	bStn3MegasonicOnOffLevel[1]:=FALSE;
	bStn3MegasonicOnOffLevel[2]:=FALSE;
	bStn3MegasonicOnOffLevel[4]:=FALSE;
	bStn3MegasonicOnOffLevel[5]:=FALSE;
END_IF

bResetMegasonicPower_RE[4](CLK:=bStn3MegasonicOnOffLevel[4]  , Q=> );	
IF bResetMegasonicPower_RE[4].Q THEN
	ARwDO[eY11104_Stn03MegasonicGenerator01Power01].15 :=FALSE;
	ARwDO[eY11105_Stn03MegasonicGenerator01Power02].15 :=FALSE;
	ARwDO[eY11106_Stn03MegasonicGenerator01Power03].15 :=FALSE;
	ARwDO[eY11108_Stn03MegasonicGenerator01Power05].15 :=FALSE;
	
	ARwDO[eY11110_Stn03MegasonicGenerator02Power01].15 :=FALSE;
	ARwDO[eY11111_Stn03MegasonicGenerator02Power02].15 :=FALSE;
	ARwDO[eY11112_Stn03MegasonicGenerator02Power03].15 :=FALSE;
	ARwDO[eY11114_Stn03MegasonicGenerator02Power05].15 :=FALSE;
	
	bStn3MegasonicOnOffLevel[1]:=FALSE;
	bStn3MegasonicOnOffLevel[2]:=FALSE;
	bStn3MegasonicOnOffLevel[3]:=FALSE;
	bStn3MegasonicOnOffLevel[5]:=FALSE;
END_IF

bResetMegasonicPower_RE[5](CLK:=bStn3MegasonicOnOffLevel[5]  , Q=> );	
IF bResetMegasonicPower_RE[5].Q THEN
	ARwDO[eY11104_Stn03MegasonicGenerator01Power01].15 :=FALSE;
	ARwDO[eY11105_Stn03MegasonicGenerator01Power02].15 :=FALSE;
	ARwDO[eY11106_Stn03MegasonicGenerator01Power03].15 :=FALSE;
	ARwDO[eY11107_Stn03MegasonicGenerator01Power04].15 :=FALSE;
	
	ARwDO[eY11110_Stn03MegasonicGenerator02Power01].15 :=FALSE;
	ARwDO[eY11111_Stn03MegasonicGenerator02Power02].15 :=FALSE;
	ARwDO[eY11112_Stn03MegasonicGenerator02Power03].15 :=FALSE;
	ARwDO[eY11107_Stn03MegasonicGenerator01Power04].15 :=FALSE;
	
	bStn3MegasonicOnOffLevel[1]:=FALSE;
	bStn3MegasonicOnOffLevel[2]:=FALSE;
	bStn3MegasonicOnOffLevel[3]:=FALSE;
	bStn3MegasonicOnOffLevel[4]:=FALSE;
END_IF	


//////// Station 6 Megasonic 
bResetMegasonicPower_RE[6](CLK:=bStn6MegasonicOnOffLevel[1]  , Q=> );	
IF bResetMegasonicPower_RE[6].Q THEN
	ARwDO[eY12004_Stn06MegasonicGenerator01Power02].15 :=FALSE;
	ARwDO[eY12005_Stn06MegasonicGenerator01Power03].15 :=FALSE;
	ARwDO[eY12006_Stn06MegasonicGenerator01Power04].15 :=FALSE;
	ARwDO[eY12007_Stn06MegasonicGenerator01Power05].15 :=FALSE;
	
	ARwDO[eY12010_Stn06MegasonicGenerator02Power02].15 :=FALSE;
	ARwDO[eY12011_Stn06MegasonicGenerator02Power03].15 :=FALSE;
	ARwDO[eY12012_Stn06MegasonicGenerator02Power04].15 :=FALSE;
	ARwDO[eY12013_Stn06MegasonicGenerator02Power05].15 :=FALSE;
	
	bStn6MegasonicOnOffLevel[2] := FALSE;
	bStn6MegasonicOnOffLevel[3] := FALSE;
	bStn6MegasonicOnOffLevel[4] := FALSE;
	bStn6MegasonicOnOffLevel[5] := FALSE;
	
END_IF

bResetMegasonicPower_RE[7](CLK:=bStn6MegasonicOnOffLevel[2]  , Q=> );	
IF bResetMegasonicPower_RE[7].Q THEN
	ARwDO[eY12003_Stn06MegasonicGenerator01Power01].15 :=FALSE;
	ARwDO[eY12005_Stn06MegasonicGenerator01Power03].15 :=FALSE;
	ARwDO[eY12006_Stn06MegasonicGenerator01Power04].15 :=FALSE;
	ARwDO[eY12007_Stn06MegasonicGenerator01Power05].15 :=FALSE;
	
	ARwDO[eY12009_Stn06MegasonicGenerator02Power01].15 :=FALSE;
	ARwDO[eY12011_Stn06MegasonicGenerator02Power03].15 :=FALSE;
	ARwDO[eY12012_Stn06MegasonicGenerator02Power04].15 :=FALSE;
	ARwDO[eY12013_Stn06MegasonicGenerator02Power05].15 :=FALSE;
	
	bStn6MegasonicOnOffLevel[1] := FALSE;
	bStn6MegasonicOnOffLevel[3] := FALSE;
	bStn6MegasonicOnOffLevel[4] := FALSE;
	bStn6MegasonicOnOffLevel[5] := FALSE;
END_IF
	
	


bResetMegasonicPower_RE[8](CLK:=bStn6MegasonicOnOffLevel[3]  , Q=> );	
IF bResetMegasonicPower_RE[8].Q THEN
	ARwDO[eY12003_Stn06MegasonicGenerator01Power01].15 :=FALSE;
	ARwDO[eY12004_Stn06MegasonicGenerator01Power02].15 :=FALSE;
	ARwDO[eY12006_Stn06MegasonicGenerator01Power04].15 :=FALSE;
	ARwDO[eY12007_Stn06MegasonicGenerator01Power05].15 :=FALSE;
	
	ARwDO[eY12009_Stn06MegasonicGenerator02Power01].15 :=FALSE;
	ARwDO[eY12010_Stn06MegasonicGenerator02Power02].15 :=FALSE;
	ARwDO[eY12012_Stn06MegasonicGenerator02Power04].15 :=FALSE;
	ARwDO[eY12013_Stn06MegasonicGenerator02Power05].15 :=FALSE;
	
	bStn6MegasonicOnOffLevel[1] := FALSE;
	bStn6MegasonicOnOffLevel[2] := FALSE;
	bStn6MegasonicOnOffLevel[4] := FALSE;
	bStn6MegasonicOnOffLevel[5] := FALSE;
END_IF

	

bResetMegasonicPower_RE[9](CLK:=bStn6MegasonicOnOffLevel[4]  , Q=> );	
IF bResetMegasonicPower_RE[9].Q THEN
	ARwDO[eY12003_Stn06MegasonicGenerator01Power01].15 :=FALSE;
	ARwDO[eY12004_Stn06MegasonicGenerator01Power02].15 :=FALSE;
	ARwDO[eY12005_Stn06MegasonicGenerator01Power03].15 :=FALSE;
	ARwDO[eY12007_Stn06MegasonicGenerator01Power05].15 :=FALSE;
	
	ARwDO[eY12009_Stn06MegasonicGenerator02Power01].15 :=FALSE;
	ARwDO[eY12010_Stn06MegasonicGenerator02Power02].15 :=FALSE;
	ARwDO[eY12011_Stn06MegasonicGenerator02Power03].15 :=FALSE;
	ARwDO[eY12013_Stn06MegasonicGenerator02Power05].15 :=FALSE;
	
	bStn6MegasonicOnOffLevel[1] := FALSE;
	bStn6MegasonicOnOffLevel[2] := FALSE;
	bStn6MegasonicOnOffLevel[3] := FALSE;
	bStn6MegasonicOnOffLevel[5] := FALSE;
END_IF

bResetMegasonicPower_RE[10](CLK:=bStn6MegasonicOnOffLevel[5]  , Q=> );	
IF bResetMegasonicPower_RE[10].Q THEN
	ARwDO[eY12003_Stn06MegasonicGenerator01Power01].15 :=FALSE;
	ARwDO[eY12004_Stn06MegasonicGenerator01Power02].15 :=FALSE;
	ARwDO[eY12005_Stn06MegasonicGenerator01Power03].15 :=FALSE;
	ARwDO[eY12006_Stn06MegasonicGenerator01Power04].15 :=FALSE;
	
	ARwDO[eY12009_Stn06MegasonicGenerator02Power01].15 :=FALSE;
	ARwDO[eY12010_Stn06MegasonicGenerator02Power02].15 :=FALSE;
	ARwDO[eY12011_Stn06MegasonicGenerator02Power03].15 :=FALSE;
	ARwDO[eY12012_Stn06MegasonicGenerator02Power04].15 :=FALSE;
	
	bStn6MegasonicOnOffLevel[1] := FALSE;
	bStn6MegasonicOnOffLevel[2] := FALSE;
	bStn6MegasonicOnOffLevel[3] := FALSE;
	bStn6MegasonicOnOffLevel[4] := FALSE;
END_IF
END_ACTION

END_PROGRAM

// ---- POUs/MainProgram/ManualCtrl/ManualCtrl.TcPOU
PROGRAM ManualCtrl
VAR

	Manual1PageEnable: BOOL;
	Manual2PageEnable: BOOL;
	MPAGE1: MANUAL_PAGE;
	MPAGE2: MANUAL_PAGE;

END_VAR

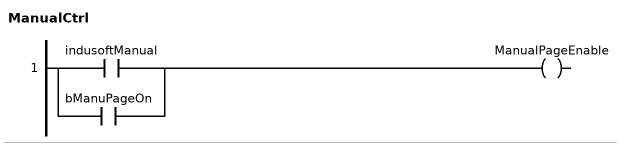
// NETWORK 1
ManualPageEnable := indusoftManual OR bManuPageOn;

END_PROGRAM

// ---- FBs/B_JKS_OldFB/Compare/MANUAL_PAGE.TcPOU
FUNCTION_BLOCK MANUAL_PAGE
VAR_INPUT
	STRING_PG1 : STRING;
	STRING_PG2 : STRING;
	STRING_PG3 : STRING;
	STRING_PG4 : STRING;
	STRING_PG5 : STRING;
	STRING_PG6 : STRING;
	STRING_PG7 : STRING;
	STRING_PG8 : STRING;
	STRING_PG9 : STRING;
	STRING_PG10 : STRING;
	STRING_PG11 : STRING;
	STRING_PG12 : STRING;
	STRING_PG13 : STRING;
	STRING_PG14 : STRING;
	STRING_PG15 : STRING;
	STRING_PG16 : STRING;
	STRING_PG17 : STRING;
	STRING_PG18 : STRING;
	STRING_PG19 : STRING;
	STRING_PG20 : STRING;
	STRING_CVISU : STRING;


END_VAR
VAR_OUTPUT
	PG_CONFIRMED_BOOL : BOOL;

END_VAR
VAR
END_VAR

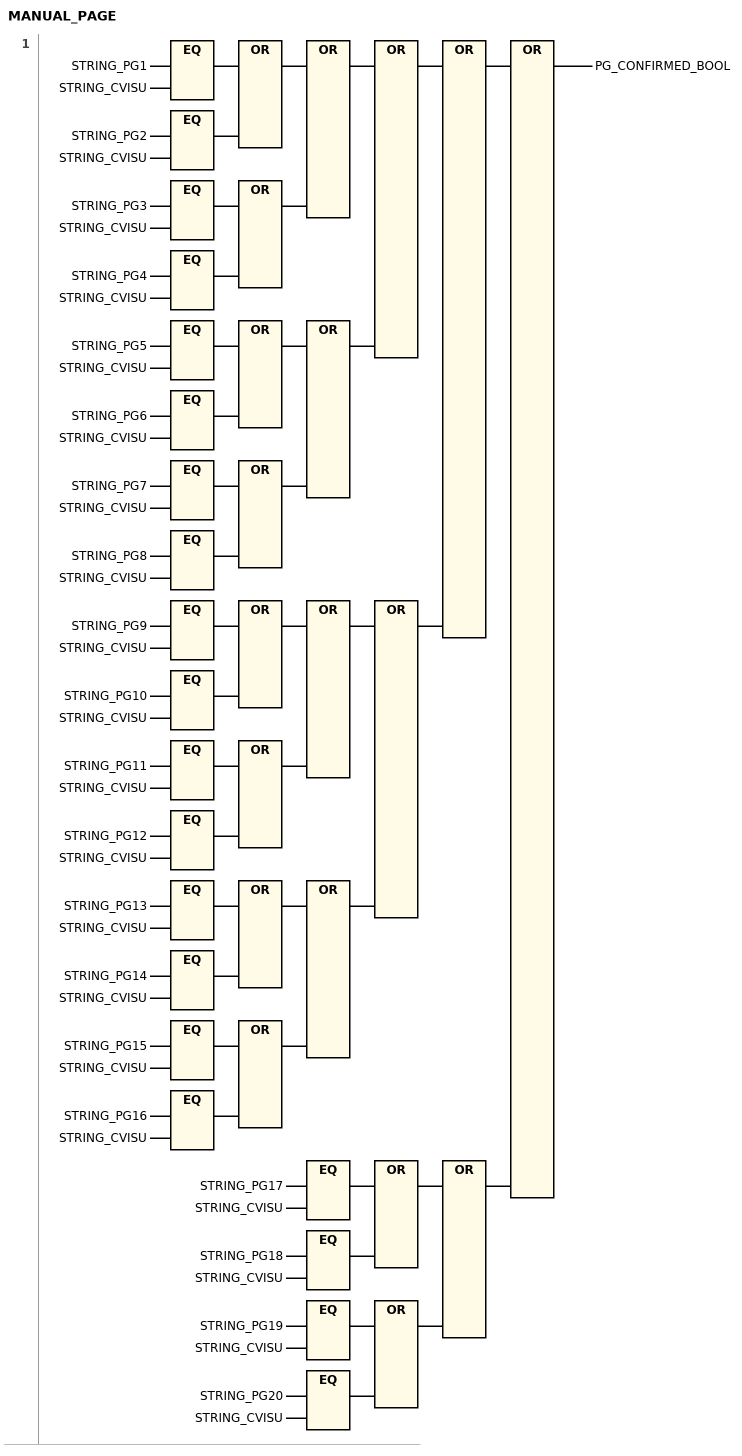
// NETWORK 1
PG_CONFIRMED_BOOL := ((((STRING_PG1 = STRING_CVISU OR STRING_PG2 = STRING_CVISU) OR (STRING_PG3 = STRING_CVISU OR STRING_PG4 = STRING_CVISU)) OR ((STRING_PG5 = STRING_CVISU OR STRING_PG6 = STRING_CVISU) OR (STRING_PG7 = STRING_CVISU OR STRING_PG8 = STRING_CVISU))) OR (((STRING_PG9 = STRING_CVISU OR STRING_PG10 = STRING_CVISU) OR (STRING_PG11 = STRING_CVISU OR STRING_PG12 = STRING_CVISU)) OR ((STRING_PG13 = STRING_CVISU OR STRING_PG14 = STRING_CVISU) OR (STRING_PG15 = STRING_CVISU OR STRING_PG16 = STRING_CVISU)))) OR ((STRING_PG17 = STRING_CVISU OR STRING_PG18 = STRING_CVISU) OR (STRING_PG19 = STRING_CVISU OR STRING_PG20 = STRING_CVISU));

END_FUNCTION_BLOCK

// ---- POUs/MainProgram/ManualCtrl/ManualCtrl_Arm.TcPOU
PROGRAM ManualCtrl_Arm
VAR
END_VAR

(*=================================Station Unhook Position================================*)
(*xxxxxxxxxx ARM 1 xxxxxxxxxx*)
IF ARDSArmCtrl[1].AR3sbPositionCfm[2,1,7] THEN
	bArm1HorzLD1Unhook_30			:= FALSE;
END_IF

IF ARDSArmCtrl[1].AR3sbPositionCfm[3,1,7] THEN
	bArm1HorzULD1Unhook_30		:= FALSE;
END_IF

IF ARDSArmCtrl[1].AR3sbPositionCfm[1,1,7] THEN
	bArm1HorzStn1Unhook_30			:= FALSE;
END_IF

IF ARDSArmCtrl[1].AR3sbPositionCfm[1,2,7] THEN
	bArm1HorzStn2Unhook_30			:= FALSE;
END_IF

IF ARDSArmCtrl[1].AR3sbPositionCfm[1,3,7] THEN
	bArm1HorzStn3Unhook_30			:= FALSE;
END_IF

IF ARDSArmCtrl[1].AR3sbPositionCfm[1,4,7] THEN
	bArm1HorzStn4Unhook_30			:= FALSE;
END_IF

IF ARDSArmCtrl[1].AR3sbPositionCfm[1,5,7] THEN
	bArm1HorzStn5Unhook_30			:= FALSE;
END_IF

IF ARDSArmCtrl[1].AR3sbPositionCfm[1,6,7] THEN
	bArm1HorzStn6Unhook_30			:= FALSE;
END_IF

IF ARDSArmCtrl[1].AR3sbPositionCfm[1,7,7] THEN
	bArm1HorzStn7Unhook_30			:= FALSE;
END_IF

IF ARDSArmCtrl[1].AR3sbPositionCfm[1,8,7] THEN
	bArm1HorzStn8Unhook_30			:= FALSE;
END_IF

IF ARDSArmCtrl[1].AR3sbPositionCfm[1,9,7] THEN
	bArm1HorzStn9Unhook_30			:= FALSE;
END_IF

IF ARDSArmCtrl[1].AR3sbPositionCfm[1,10,7] THEN
	bArm1HorzStn10Unhook_30		:= FALSE;
END_IF

IF ARDSArmCtrl[1].AR3sbPositionCfm[1,11,7] THEN
	bArm1HorzStn11Unhook_30		:= FALSE;
END_IF

IF ARDSArmCtrl[1].AR3sbPositionCfm[1,12,7] THEN
	bArm1HorzStn12Unhook_30		:= FALSE;
END_IF

(*xxxxxxxxxx ARM 2 xxxxxxxxxx*)
IF ARDSArmCtrl[2].AR3sbPositionCfm[2,1,7] THEN
	bArm2HorzLD1Unhook_30			:= FALSE;
END_IF

IF ARDSArmCtrl[2].AR3sbPositionCfm[3,1,7] THEN
	bArm2HorzULD1Unhook_30		:= FALSE;
END_IF

IF ARDSArmCtrl[2].AR3sbPositionCfm[1,1,7] THEN
	bArm2HorzStn1Unhook_30			:= FALSE;
END_IF

IF ARDSArmCtrl[2].AR3sbPositionCfm[1,2,7] THEN
	bArm2HorzStn2Unhook_30			:= FALSE;
END_IF

IF ARDSArmCtrl[2].AR3sbPositionCfm[1,3,7] THEN
	bArm2HorzStn3Unhook_30			:= FALSE;
END_IF

IF ARDSArmCtrl[2].AR3sbPositionCfm[1,4,7] THEN
	bArm2HorzStn4Unhook_30			:= FALSE;
END_IF

IF ARDSArmCtrl[2].AR3sbPositionCfm[1,5,7] THEN
	bArm2HorzStn5Unhook_30			:= FALSE;
END_IF

IF ARDSArmCtrl[2].AR3sbPositionCfm[1,6,7] THEN
	bArm2HorzStn6Unhook_30			:= FALSE;
END_IF

IF ARDSArmCtrl[2].AR3sbPositionCfm[1,7,7] THEN
	bArm2HorzStn7Unhook_30			:= FALSE;
END_IF

IF ARDSArmCtrl[2].AR3sbPositionCfm[1,8,7] THEN
	bArm2HorzStn8Unhook_30			:= FALSE;
END_IF

IF ARDSArmCtrl[2].AR3sbPositionCfm[1,9,7] THEN
	bArm2HorzStn9Unhook_30			:= FALSE;
END_IF

IF ARDSArmCtrl[2].AR3sbPositionCfm[1,10,7] THEN
	bArm2HorzStn10Unhook_30		:= FALSE;
END_IF

IF ARDSArmCtrl[2].AR3sbPositionCfm[1,11,7] THEN
	bArm2HorzStn11Unhook_30		:= FALSE;
END_IF

IF ARDSArmCtrl[2].AR3sbPositionCfm[1,12,7] THEN
	bArm2HorzStn12Unhook_30		:= FALSE;
END_IF


(*=================================Station Hook Position================================*)
(*xxxxxxxxxx ARM 1 xxxxxxxxxx*)
IF ARDSArmCtrl[1].AR3sbPositionCfm[2,1,8] THEN
	bArm1HorzLD1Hook_30			:= FALSE;
END_IF

IF ARDSArmCtrl[1].AR3sbPositionCfm[3,1,8] THEN
	bArm1HorzULD1Hook_30			:= FALSE;
END_IF

IF ARDSArmCtrl[1].AR3sbPositionCfm[1,1,8] THEN
	bArm1HorzStn1Hook_30			:= FALSE;
END_IF

IF ARDSArmCtrl[1].AR3sbPositionCfm[1,2,8] THEN
	bArm1HorzStn2Hook_30			:= FALSE;
END_IF

IF ARDSArmCtrl[1].AR3sbPositionCfm[1,3,8] THEN
	bArm1HorzStn3Hook_30			:= FALSE;
END_IF

IF ARDSArmCtrl[1].AR3sbPositionCfm[1,4,8] THEN
	bArm1HorzStn4Hook_30			:= FALSE;
END_IF

IF ARDSArmCtrl[1].AR3sbPositionCfm[1,5,8] THEN
	bArm1HorzStn5Hook_30			:= FALSE;
END_IF

IF ARDSArmCtrl[1].AR3sbPositionCfm[1,6,8] THEN
	bArm1HorzStn6Hook_30			:= FALSE;
END_IF

IF ARDSArmCtrl[1].AR3sbPositionCfm[1,7,8] THEN
	bArm1HorzStn7Hook_30			:= FALSE;
END_IF

IF ARDSArmCtrl[1].AR3sbPositionCfm[1,8,8] THEN
	bArm1HorzStn8Hook_30			:= FALSE;
END_IF


IF ARDSArmCtrl[1].AR3sbPositionCfm[1,9,8] THEN
	bArm1HorzStn9Hook_30			:= FALSE;
END_IF

IF ARDSArmCtrl[1].AR3sbPositionCfm[1,10,8] THEN
	bArm1HorzStn10Hook_30			:= FALSE;
END_IF

IF ARDSArmCtrl[1].AR3sbPositionCfm[1,11,8] THEN
	bArm1HorzStn11Hook_30			:= FALSE;
END_IF

IF ARDSArmCtrl[1].AR3sbPositionCfm[1,12,8] THEN
	bArm1HorzStn12Hook_30			:= FALSE;
END_IF

(*xxxxxxxxxx ARM 2 xxxxxxxxxx*)
IF ARDSArmCtrl[2].AR3sbPositionCfm[2,1,8] THEN
	bArm2HorzLD1Hook_30			:= FALSE;
END_IF

IF ARDSArmCtrl[2].AR3sbPositionCfm[3,1,8] THEN
	bArm2HorzULD1Hook_30			:= FALSE;
END_IF

IF ARDSArmCtrl[2].AR3sbPositionCfm[1,1,8] THEN
	bArm2HorzStn1Hook_30			:= FALSE;
END_IF

IF ARDSArmCtrl[2].AR3sbPositionCfm[1,2,8] THEN
	bArm2HorzStn2Hook_30			:= FALSE;
END_IF

IF ARDSArmCtrl[2].AR3sbPositionCfm[1,3,8] THEN
	bArm2HorzStn3Hook_30			:= FALSE;
END_IF

IF ARDSArmCtrl[2].AR3sbPositionCfm[1,4,8] THEN
	bArm2HorzStn4Hook_30			:= FALSE;
END_IF

IF ARDSArmCtrl[2].AR3sbPositionCfm[1,5,8] THEN
	bArm2HorzStn5Hook_30			:= FALSE;
END_IF

IF ARDSArmCtrl[2].AR3sbPositionCfm[1,6,8] THEN
	bArm2HorzStn6Hook_30			:= FALSE;
END_IF

IF ARDSArmCtrl[2].AR3sbPositionCfm[1,7,8] THEN
	bArm2HorzStn7Hook_30			:= FALSE;
END_IF

IF ARDSArmCtrl[2].AR3sbPositionCfm[1,8,8] THEN
	bArm2HorzStn8Hook_30			:= FALSE;
END_IF


IF ARDSArmCtrl[2].AR3sbPositionCfm[1,9,8] THEN
	bArm2HorzStn9Hook_30			:= FALSE;
END_IF

IF ARDSArmCtrl[2].AR3sbPositionCfm[1,10,8] THEN
	bArm2HorzStn10Hook_30			:= FALSE;
END_IF

IF ARDSArmCtrl[2].AR3sbPositionCfm[1,11,8] THEN
	bArm2HorzStn11Hook_30			:= FALSE;
END_IF

IF ARDSArmCtrl[2].AR3sbPositionCfm[1,12,8] THEN
	bArm2HorzStn12Hook_30			:= FALSE;
END_IF


(*=================================Station Up / Down Position================================*)
(*xxxxxxxxxx ARM 1 xxxxxxxxxx*)
IF ARDSArmCtrl[1].AR3sbPositionCfm[2,1,1] OR NOT ARbArmVertHomeDone[1] THEN
	bArm1VertLD1Up_30				:= FALSE;
END_IF

IF ARDSArmCtrl[1].AR3sbPositionCfm[2,1,6] THEN
	bArm1VertLD1Down_30			:= FALSE;
END_IF

IF ARDSArmCtrl[1].AR3sbPositionCfm[3,1,6] THEN
	 bArm1VertULD1Down_30 			:= FALSE;
END_IF

IF ARDSArmCtrl[1].AR3sbPositionCfm[1,1,6] THEN
	bArm1VertStn1Down_30			:= FALSE;
END_IF

IF ARDSArmCtrl[1].AR3sbPositionCfm[1,2,6] THEN
	bArm1VertStn2Down_30			:= FALSE;
END_IF

IF ARDSArmCtrl[1].AR3sbPositionCfm[1,3,6] THEN
	bArm1VertStn3Down_30			:= FALSE;
END_IF

IF ARDSArmCtrl[1].AR3sbPositionCfm[1,4,6] THEN
	bArm1VertStn4Down_30			:= FALSE;
END_IF

IF ARDSArmCtrl[1].AR3sbPositionCfm[1,5,6] THEN
	bArm1VertStn5Down_30			:= FALSE;
END_IF

IF ARDSArmCtrl[1].AR3sbPositionCfm[1,6,6] THEN
	bArm1VertStn6Down_30			:= FALSE;
END_IF

IF ARDSArmCtrl[1].AR3sbPositionCfm[1,7,6] THEN
	bArm1VertStn7Down_30			:= FALSE;
END_IF

IF ARDSArmCtrl[1].AR3sbPositionCfm[1,8,6] THEN
	bArm1VertStn8Down_30			:= FALSE;
END_IF

IF ARDSArmCtrl[1].AR3sbPositionCfm[1,9,6] THEN
	bArm1VertStn9Down_30			:= FALSE;
END_IF

IF ARDSArmCtrl[1].AR3sbPositionCfm[1,10,6] THEN
	bArm1VertStn10Down_30			:= FALSE;
END_IF

IF ARDSArmCtrl[1].AR3sbPositionCfm[1,11,6] THEN
	bArm1VertStn11Down_30			:= FALSE;
END_IF

IF ARDSArmCtrl[1].AR3sbPositionCfm[1,12,6] THEN
	bArm1VertStn12Down_30			:= FALSE;
END_IF

(*xxxxxxxxxx ARM 2 xxxxxxxxxx*)
IF ARDSArmCtrl[2].AR3sbPositionCfm[3,1,1] OR NOT ARbArmVertHomeDone[2] THEN
	bArm2VertULD1Up_30				:= FALSE;
END_IF

IF ARDSArmCtrl[2].AR3sbPositionCfm[2,1,6] THEN
	bArm2VertLD1Down_30			:= FALSE;
END_IF

IF ARDSArmCtrl[2].AR3sbPositionCfm[3,1,6] THEN
	 bArm2VertULD1Down_30 			:= FALSE;
END_IF

IF ARDSArmCtrl[2].AR3sbPositionCfm[1,1,6] THEN
	bArm2VertStn1Down_30			:= FALSE;
END_IF

IF ARDSArmCtrl[2].AR3sbPositionCfm[1,2,6] THEN
	bArm2VertStn2Down_30			:= FALSE;
END_IF

IF ARDSArmCtrl[2].AR3sbPositionCfm[1,3,6] THEN
	bArm2VertStn3Down_30			:= FALSE;
END_IF

IF ARDSArmCtrl[2].AR3sbPositionCfm[1,4,6] THEN
	bArm2VertStn4Down_30			:= FALSE;
END_IF

IF ARDSArmCtrl[2].AR3sbPositionCfm[1,5,6] THEN
	bArm2VertStn5Down_30			:= FALSE;
END_IF

IF ARDSArmCtrl[2].AR3sbPositionCfm[1,6,6] THEN
	bArm2VertStn6Down_30			:= FALSE;
END_IF

IF ARDSArmCtrl[2].AR3sbPositionCfm[1,7,6] THEN
	bArm2VertStn7Down_30			:= FALSE;
END_IF

IF ARDSArmCtrl[2].AR3sbPositionCfm[1,8,6] THEN
	bArm2VertStn8Down_30			:= FALSE;
END_IF

IF ARDSArmCtrl[2].AR3sbPositionCfm[1,9,6] THEN
	bArm2VertStn9Down_30			:= FALSE;
END_IF

IF ARDSArmCtrl[2].AR3sbPositionCfm[1,10,6] THEN
	bArm2VertStn10Down_30			:= FALSE;
END_IF

IF ARDSArmCtrl[2].AR3sbPositionCfm[1,11,6] THEN
	bArm2VertStn11Down_30			:= FALSE;
END_IF

IF ARDSArmCtrl[2].AR3sbPositionCfm[1,12,6] THEN
	bArm2VertStn12Down_30			:= FALSE;
END_IF


(*=================================Station Slow Pull Position================================*)


IF ARDSArmCtrl[1].AR3sbPositionCfm[1,9,2] THEN      (*Stn 9 SlowPull Mid Down*)
	bArm1VertStn9SpSlanted_30		:= FALSE;
END_IF


IF bArmSlowPullUpCFM OR NOT ARbArmSlowPullHomeDone[1] THEN
	bSlowPull1LifterStn9Up_30			:= FALSE;
END_IF


IF bArmSlowPullDownCFM OR NOT ARbArmSlowPullHomeDone[1] THEN
	bSlowPull1LifterStn9Down_30		:= FALSE;
END_IF


(*=================================Station Position================================*)

IF EmergencyStop OR NOT ManualPageEnable THEN

	bArm1VertHomeStart_30			:= FALSE;
	bArm1HorzHomeStart_30			:= FALSE;
	bSlowPull1LifterHomeStart_30		:= FALSE;

	bArm2VertHomeStart_30			:= FALSE;
	bArm2HorzHomeStart_30			:= FALSE;
	bSlowPull2LifterHomeStart_30		:= FALSE;

	bArm1HorzLD1Unhook_30			:= FALSE;
	bArm1HorzULD1Unhook_30		:= FALSE;
	bArm1HorzStn1Unhook_30 			:= FALSE;
	bArm1HorzStn2Unhook_30			:= FALSE;
	bArm1HorzStn3Unhook_30			:= FALSE;
	bArm1HorzStn4Unhook_30			:= FALSE;
	bArm1HorzStn5Unhook_30 			:= FALSE;
	bArm1HorzStn6Unhook_30			:= FALSE;
	bArm1HorzStn7Unhook_30			:= FALSE;
	bArm1HorzStn8Unhook_30			:= FALSE;
	bArm1HorzStn9Unhook_30 			:= FALSE;
	bArm1HorzStn10Unhook_30		:= FALSE;
	bArm1HorzStn11Unhook_30		:= FALSE;
	bArm1HorzStn12Unhook_30		:= FALSE;

	bArm2HorzLD1Unhook_30			:= FALSE;
	bArm2HorzULD1Unhook_30		:= FALSE;
	bArm2HorzStn1Unhook_30 			:= FALSE;
	bArm2HorzStn2Unhook_30			:= FALSE;
	bArm2HorzStn3Unhook_30			:= FALSE;
	bArm2HorzStn4Unhook_30			:= FALSE;
	bArm2HorzStn5Unhook_30 			:= FALSE;
	bArm2HorzStn6Unhook_30			:= FALSE;
	bArm2HorzStn7Unhook_30			:= FALSE;
	bArm2HorzStn8Unhook_30			:= FALSE;
	bArm2HorzStn9Unhook_30 			:= FALSE;
	bArm2HorzStn10Unhook_30		:= FALSE;
	bArm2HorzStn11Unhook_30		:= FALSE;
	bArm2HorzStn12Unhook_30		:= FALSE;

	bArm1HorzLD1Hook_30			:= FALSE;
	bArm1HorzULD1Hook_30			:= FALSE;
	bArm1HorzStn1Hook_30			:= FALSE;
	bArm1HorzStn2Hook_30			:= FALSE;
	bArm1HorzStn3Hook_30			:= FALSE;
	bArm1HorzStn4Hook_30			:= FALSE;
	bArm1HorzStn5Hook_30			:= FALSE;
	bArm1HorzStn6Hook_30			:= FALSE;
	bArm1HorzStn7Hook_30			:= FALSE;
	bArm1HorzStn8Hook_30			:= FALSE;
	bArm1HorzStn9Hook_30			:= FALSE;
	bArm1HorzStn10Hook_30			:= FALSE;
	bArm1HorzStn11Hook_30			:= FALSE;
	bArm1HorzStn12Hook_30			:= FALSE;

	bArm2HorzLD1Hook_30			:= FALSE;
	bArm2HorzULD1Hook_30			:= FALSE;
	bArm2HorzStn1Hook_30			:= FALSE;
	bArm2HorzStn2Hook_30			:= FALSE;
	bArm2HorzStn3Hook_30			:= FALSE;
	bArm2HorzStn4Hook_30			:= FALSE;
	bArm2HorzStn5Hook_30			:= FALSE;
	bArm2HorzStn6Hook_30			:= FALSE;
	bArm2HorzStn7Hook_30			:= FALSE;
	bArm2HorzStn8Hook_30			:= FALSE;
	bArm2HorzStn9Hook_30			:= FALSE;
	bArm2HorzStn10Hook_30			:= FALSE;
	bArm2HorzStn11Hook_30			:= FALSE;
	bArm2HorzStn12Hook_30			:= FALSE;

	bArm1VertLD1Up_30				:= FALSE;
	bArm1VertLD1Up_28 				:= FALSE;

	bArm2VertULD1Up_30				:= FALSE;
	bArm2VertULD1Up_28 				:= FALSE;

	bArm1VertLD1Down_30			:= FALSE;
	bArm1VertULD1Down_30			:= FALSE;
	bArm1VertStn1Down_30			:= FALSE;
	bArm1VertStn2Down_30			:= FALSE;
	bArm1VertStn3Down_30			:= FALSE;
	bArm1VertStn4Down_30			:= FALSE;
	bArm1VertStn5Down_30			:= FALSE;
	bArm1VertStn6Down_30			:= FALSE;
	bArm1VertStn7Down_30			:= FALSE;
	bArm1VertStn8Down_30			:= FALSE;
	bArm1VertStn9Down_30			:= FALSE;
	bArm1VertStn10Down_30			:= FALSE;

	bArm2VertLD1Down_30			:= FALSE;
	bArm2VertULD1Down_30			:= FALSE;
	bArm2VertStn1Down_30			:= FALSE;
	bArm2VertStn2Down_30			:= FALSE;
	bArm2VertStn3Down_30			:= FALSE;
	bArm2VertStn4Down_30			:= FALSE;
	bArm2VertStn5Down_30			:= FALSE;
	bArm2VertStn6Down_30			:= FALSE;
	bArm2VertStn7Down_30			:= FALSE;
	bArm2VertStn8Down_30			:= FALSE;
	bArm2VertStn9Down_30			:= FALSE;
	bArm2VertStn10Down_30			:= FALSE;

	bArm1VertStn9SpSlanted_30		:= FALSE;
	bArm2VertStn9SpSlanted_30		:= FALSE;

	bArm1VertStn10SpSlanted_30		:= FALSE;
	bArm2VertStn10SpSlanted_30		:= FALSE;

	bSlowPull1LifterStn9Up_30			:= FALSE;
	bSlowPull1LifterStn9Down_30		:= FALSE;

	bSlowPull1LifterStn10Up_30			:= FALSE;
	bSlowPull1LifterStn10Down_30		:= FALSE;

	bSlowPull2LifterStn10Up_30			:= FALSE;
	bSlowPull2LifterStn10Down_30		:= FALSE;

	bManualArmHome				:= FALSE;

END_IF


IF ARbArmVertHomeDone[1] THEN
	bArm1VertHomeStart_30			:= FALSE;
END_IF

IF ARbArmHorzHomeDone[1] THEN
	bArm1HorzHomeStart_30			:= FALSE;
END_IF

IF ARbArmSlowPullHomeDone[1] THEN
	bSlowPull1LifterHomeStart_30		:= FALSE;
END_IF


IF ARbArmVertHomeDone[2] THEN
	bArm2VertHomeStart_30			:= FALSE;
END_IF

IF ARbArmHorzHomeDone[2] THEN
	bArm2HorzHomeStart_30			:= FALSE;
END_IF


IF ARbArmVertHomeDone[1] AND ARbArmHorzHomeDone[1] THEN
	bManualArmHome				:= FALSE;
END_IF

IF bManualArmHome AND ARbArmVertHomeDone[1] AND NOT ARDSArmCtrl[1].AR3sbPositionCfm[2,1,1] THEN
bArm1VertLD1Up_28 					:= TRUE;
ELSE
bArm1VertLD1Up_28 					:= FALSE;
END_IF

END_PROGRAM

// ---- POUs/MainProgram/ManualCtrl/ManualLifterJog.TcPOU
 PROGRAM ManualLifterJog
VAR
	ArmSlowPullJogCtrlFB: MC_Jog;
END_VAR

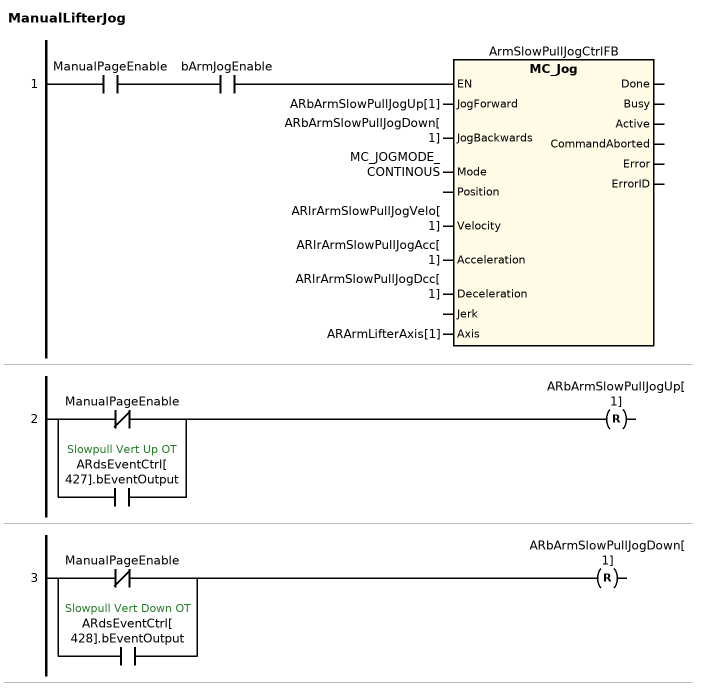
// NETWORK 1
IF ManualPageEnable AND bArmJogEnable THEN
    ArmSlowPullJogCtrlFB(
        JogForward := ARbArmSlowPullJogUp[1],
        JogBackwards := ARbArmSlowPullJogDown[1],
        Mode := MC_JOGMODE_CONTINOUS,
        Velocity := ARlrArmSlowPullJogVelo[1],
        Acceleration := ARlrArmSlowPullJogAcc[1],
        Deceleration := ARlrArmSlowPullJogDcc[1],
        Axis := ARArmLifterAxis[1]); // MC_Jog
END_IF

// NETWORK 2
//   ARdsEventCtrl[427].bEventOutput: Slowpull Vert Up OT
ARbArmSlowPullJogUp[1] R= NOT ManualPageEnable OR ARdsEventCtrl[427].bEventOutput;

// NETWORK 3
//   ARdsEventCtrl[428].bEventOutput: Slowpull Vert Down OT
ARbArmSlowPullJogDown[1] R= NOT ManualPageEnable OR ARdsEventCtrl[428].bEventOutput;

END_PROGRAM

// ---- POUs/MainProgram/Other/ArmXYPosAdjust.TcPOU
PROGRAM ArmXYPosAdjust
VAR
	fbHMISimulateArmMovement_Arm1: fbHMISimulateArmMovement;
	fbHMISimulateArmMovement_Arm2: fbHMISimulateArmMovement;
	dummy2: LREAL;
	dummy1: LREAL;
END_VAR

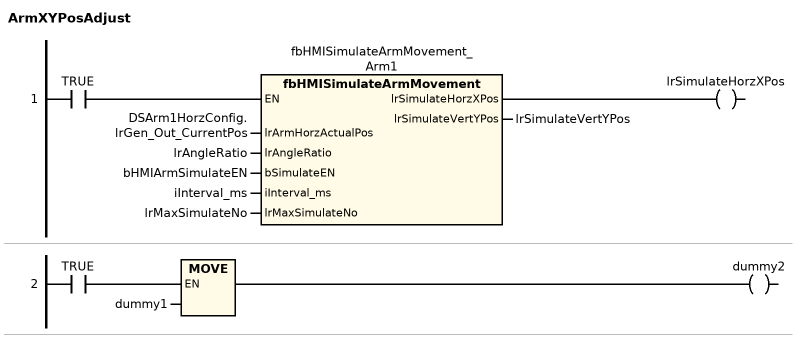
// NETWORK 1
fbHMISimulateArmMovement_Arm1(
    lrArmHorzActualPos := DSArm1HorzConfig.lrGen_Out_CurrentPos,
    lrAngleRatio := lrAngleRatio,
    bSimulateEN := bHMIArmSimulateEN,
    iInterval_ms := iInterval_ms,
    lrMaxSimulateNo := lrMaxSimulateNo,
    lrSimulateVertYPos => lrSimulateVertYPos); // fbHMISimulateArmMovement
lrSimulateHorzXPos := fbHMISimulateArmMovement_Arm1.lrSimulateHorzXPos;

// NETWORK 2
dummy2 := dummy1;

END_PROGRAM

// ---- FBs/B_JKS_NewFB/FBP-HMI/fbHMISimulateArmMovement.TcPOU
FUNCTION_BLOCK fbHMISimulateArmMovement
VAR_INPUT
	lrArmHorzActualPos : LREAL;
	lrAngleRatio : LREAL;
	bSimulateEN : BOOL;
	iInterval_ms : INT;
	lrMaxSimulateNo : LREAL;


END_VAR
VAR_OUTPUT
	lrSimulateHorzXPos : LREAL;
	lrSimulateVertYPos : LREAL;

END_VAR
VAR
	tDelayOn: TON;
	tDelayOnRE: R_TRIG;
	lrSimArmHorzActualPos: LREAL;
	bReverseCount: BOOL;
END_VAR

IF bSimulateEN THEN
	IF lrSimArmHorzActualPos > 0 AND lrAngleRatio >0 THEN
	lrSimulateHorzXPos := lrSimArmHorzActualPos;
	lrSimulateVertYPos := lrSimArmHorzActualPos * lrAngleRatio;
	ELSE
		lrSimulateHorzXPos := 0;
		lrSimulateVertYPos := 0;
	END_IF
ELSE
	IF lrArmHorzActualPos > 0 AND lrAngleRatio >0 THEN
	lrSimulateHorzXPos := lrArmHorzActualPos;
	lrSimulateVertYPos := lrArmHorzActualPos * lrAngleRatio;
	ELSE
		lrSimulateHorzXPos := 0;
		lrSimulateVertYPos := 0;
	END_IF
END_IF




(*Simulation*)


tDelayOn(IN:=NOT tDelayOn.Q , PT:=INT_TO_TIME(iInterval_ms) , Q=> , ET=> );
tDelayOnRE(CLK:=tDelayOn.Q , Q=> );

IF bSimulateEN THEN
	IF lrSimArmHorzActualPos >= lrMaxSimulateNo THEN
	bReverseCount := TRUE;
	END_IF
	
	IF  lrSimArmHorzActualPos <= 0 THEN
	bReverseCount := FALSE;
	END_IF

	IF  tDelayOnRE.Q AND NOT bReverseCount AND lrMaxSimulateNo > 0 THEN
	lrSimArmHorzActualPos := lrSimArmHorzActualPos +1;
	END_IF
	
	IF  tDelayOnRE.Q AND bReverseCount THEN
	lrSimArmHorzActualPos := lrSimArmHorzActualPos -1;
	END_IF
END_IF


IF NOT bSimulateEN THEN
bReverseCount := FALSE;
lrSimArmHorzActualPos := 0;
END_IF

END_FUNCTION_BLOCK

// ---- POUs/MainProgram/Other/BeckhoffHMIMapping.TcPOU
PROGRAM BeckhoffHMIMapping
VAR
	(*ARfbHMIAddMappingBool : ARRAY [1..500 ] OF fbHMIAddMappingBool;*)
	(*ARfbHMIAddMappingInt : ARRAY [1..500 ] OF fbHMIAddMappingInt;*)
	(*ARfbHMIAddMappingReal : ARRAY [1..500 ] OF fbHMIAddMappingReal;*)
	ARfbHMIAddMappingLreal : ARRAY [1..100 ] OF fbHMIAddMappingLreal;
	(*ARfbHMIAddMappingString : ARRAY [1..500 ] OF fbHMIAddMappingString;*)
	ARfbHMIAddMappingInt_Word : ARRAY [1..100 ] OF fbHMIAddMappingInt_Word;
	(*fbHMIAddMappingReal_Int : ARRAY [1..100] OF fbHMIAddMappingReal_Int;*)
	ARfbHMIAddMappingReal_Word : ARRAY [1..100 ] OF fbHMIAddMappingReal_Word;

	(*ARfbHMIAddMappingBoolForManual : ARRAY [1..500 ] OF fbHMIAddMappingBoolForManual;*)
	(*ARfbHMIAddMappingDWordToBoolForManual : ARRAY [1..iArmQty ] OF fbHMIAddMappingDWordToBoolForManual;*)

	(*ARfbHMIAddMappingArrayInt : ARRAY [1..10 ] OF fbHMIAddMappingArrayInt;*)
	(*ARfbHMIAddMappingArrayBool : ARRAY [1..10 ] OF fbHMIAddMappingArrayBool;*)
	(*ARfbHMIAddMappingArrayReal : ARRAY [1..10 ] OF fbHMIAddMappingArrayReal;*)
	(*ARfbHMIAddMappingArrayLreal : ARRAY [0..10 ] OF fbHMIAddMappingArrayLreal;*)
	(*ARfbHMIAddMappingArrayBool : ARRAY [1..10 ] OF fbHMIAddMappingArrayBool;*)

END_VAR

(*Loading*)

ARfbHMIAddMappingLreal[1](
bEN:=TRUE ,
ARrLrealAddress_Pro:=ARDSLdZoneHeight[1].lrTopPos,
ARrLrealAddress_Hmi:=Arm1TopPos[19]);

ARfbHMIAddMappingLreal[2](
bEN:=TRUE ,
ARrLrealAddress_Pro:=ARDSLdZoneHeight[1].lrZone1Range,
ARrLrealAddress_Hmi:=Arm1Pos1stStage[19]);

ARfbHMIAddMappingLreal[3](
bEN:=TRUE ,
ARrLrealAddress_Pro:=ARDSLdZoneHeight[1].lrZone2Range,
ARrLrealAddress_Hmi:=Arm1Pos2ndStage[19]);

ARfbHMIAddMappingLreal[4](
bEN:=TRUE ,
ARrLrealAddress_Pro:=ARDSLdZoneHeight[1].lrZone3Range,
ARrLrealAddress_Hmi:=Arm1Pos3rdStage[19]);

ARfbHMIAddMappingLreal[5](
bEN:=TRUE ,
ARrLrealAddress_Pro:=ARDSLdZoneHeight[1].lrZone4Range,
ARrLrealAddress_Hmi:=Arm1Pos4thStage[19]);

ARfbHMIAddMappingLreal[6](
bEN:=TRUE ,
ARrLrealAddress_Pro:=ARDSLdZoneHeight[1].lrBottomPos,
ARrLrealAddress_Hmi:=Arm1BottomPos[19]);

ARfbHMIAddMappingLreal[7](
bEN:=TRUE ,
ARrLrealAddress_Pro:=ARDSLdZoneHeight[1].lrMidPos,
ARrLrealAddress_Hmi:=Arm1MidPos[19]);


(*Station 1*)

ARfbHMIAddMappingLreal[8](
bEN:=TRUE ,
ARrLrealAddress_Pro:=ARDSStationZoneHeight[1].lrTopPos,
ARrLrealAddress_Hmi:=Arm1TopPos[1]);

ARfbHMIAddMappingLreal[9](
bEN:=TRUE ,
ARrLrealAddress_Pro:=ARDSStationZoneHeight[1].lrZone1Range,
ARrLrealAddress_Hmi:=Arm1Pos1stStage[1]);

ARfbHMIAddMappingLreal[10](
bEN:=TRUE ,
ARrLrealAddress_Pro:=ARDSStationZoneHeight[1].lrZone2Range,
ARrLrealAddress_Hmi:=Arm1Pos2ndStage[1]);

ARfbHMIAddMappingLreal[11](
bEN:=TRUE ,
ARrLrealAddress_Pro:=ARDSStationZoneHeight[1].lrZone3Range,
ARrLrealAddress_Hmi:=Arm1Pos3rdStage[1]);

ARfbHMIAddMappingLreal[12](
bEN:=TRUE ,
ARrLrealAddress_Pro:=ARDSStationZoneHeight[1].lrZone4Range,
ARrLrealAddress_Hmi:=Arm1Pos4thStage[1]);

ARfbHMIAddMappingLreal[13](
bEN:=TRUE ,
ARrLrealAddress_Pro:=ARDSStationZoneHeight[1].lrBottomPos,
ARrLrealAddress_Hmi:=Arm1BottomPos[1]);

ARfbHMIAddMappingLreal[14](
bEN:=TRUE ,
ARrLrealAddress_Pro:=ARDSStationZoneHeight[1].lrMidPos,
ARrLrealAddress_Hmi:=Arm1MidPos[1]);


(*Station 2*)

ARfbHMIAddMappingLreal[15](
bEN:=TRUE ,
ARrLrealAddress_Pro:=ARDSStationZoneHeight[2].lrTopPos,
ARrLrealAddress_Hmi:=Arm1TopPos[2]);

ARfbHMIAddMappingLreal[16](
bEN:=TRUE ,
ARrLrealAddress_Pro:=ARDSStationZoneHeight[2].lrZone1Range,
ARrLrealAddress_Hmi:=Arm1Pos1stStage[2]);

ARfbHMIAddMappingLreal[17](
bEN:=TRUE ,
ARrLrealAddress_Pro:=ARDSStationZoneHeight[2].lrZone2Range,
ARrLrealAddress_Hmi:=Arm1Pos2ndStage[2]);

ARfbHMIAddMappingLreal[18](
bEN:=TRUE ,
ARrLrealAddress_Pro:=ARDSStationZoneHeight[2].lrZone3Range,
ARrLrealAddress_Hmi:=Arm1Pos3rdStage[2]);

ARfbHMIAddMappingLreal[19](
bEN:=TRUE ,
ARrLrealAddress_Pro:=ARDSStationZoneHeight[2].lrZone4Range,
ARrLrealAddress_Hmi:=Arm1Pos4thStage[2]);

ARfbHMIAddMappingLreal[20](
bEN:=TRUE ,
ARrLrealAddress_Pro:=ARDSStationZoneHeight[2].lrBottomPos,
ARrLrealAddress_Hmi:=Arm1BottomPos[2]);

ARfbHMIAddMappingLreal[21](
bEN:=TRUE ,
ARrLrealAddress_Pro:=ARDSStationZoneHeight[2].lrMidPos,
ARrLrealAddress_Hmi:=Arm1MidPos[2]);


(*Station 3*)

ARfbHMIAddMappingLreal[22](
bEN:=TRUE ,
ARrLrealAddress_Pro:=ARDSStationZoneHeight[3].lrTopPos,
ARrLrealAddress_Hmi:=Arm1TopPos[3]);

ARfbHMIAddMappingLreal[23](
bEN:=TRUE ,
ARrLrealAddress_Pro:=ARDSStationZoneHeight[3].lrZone1Range,
ARrLrealAddress_Hmi:=Arm1Pos1stStage[3]);

ARfbHMIAddMappingLreal[24](
bEN:=TRUE ,
ARrLrealAddress_Pro:=ARDSStationZoneHeight[3].lrZone2Range,
ARrLrealAddress_Hmi:=Arm1Pos2ndStage[3]);

ARfbHMIAddMappingLreal[25](
bEN:=TRUE ,
ARrLrealAddress_Pro:=ARDSStationZoneHeight[3].lrZone3Range,
ARrLrealAddress_Hmi:=Arm1Pos3rdStage[3]);

ARfbHMIAddMappingLreal[26](
bEN:=TRUE ,
ARrLrealAddress_Pro:=ARDSStationZoneHeight[3].lrZone4Range,
ARrLrealAddress_Hmi:=Arm1Pos4thStage[3]);

ARfbHMIAddMappingLreal[27](
bEN:=TRUE ,
ARrLrealAddress_Pro:=ARDSStationZoneHeight[3].lrBottomPos,
ARrLrealAddress_Hmi:=Arm1BottomPos[3]);

ARfbHMIAddMappingLreal[28](
bEN:=TRUE ,
ARrLrealAddress_Pro:=ARDSStationZoneHeight[3].lrMidPos,
ARrLrealAddress_Hmi:=Arm1MidPos[3]);


(*Station 4*)

ARfbHMIAddMappingLreal[29](
bEN:=TRUE ,
ARrLrealAddress_Pro:=ARDSStationZoneHeight[4].lrTopPos,
ARrLrealAddress_Hmi:=Arm1TopPos[4]);

ARfbHMIAddMappingLreal[30](
bEN:=TRUE ,
ARrLrealAddress_Pro:=ARDSStationZoneHeight[4].lrZone1Range,
ARrLrealAddress_Hmi:=Arm1Pos1stStage[4]);

ARfbHMIAddMappingLreal[31](
bEN:=TRUE ,
ARrLrealAddress_Pro:=ARDSStationZoneHeight[4].lrZone2Range,
ARrLrealAddress_Hmi:=Arm1Pos2ndStage[4]);

ARfbHMIAddMappingLreal[32](
bEN:=TRUE ,
ARrLrealAddress_Pro:=ARDSStationZoneHeight[4].lrZone3Range,
ARrLrealAddress_Hmi:=Arm1Pos3rdStage[4]);

ARfbHMIAddMappingLreal[33](
bEN:=TRUE ,
ARrLrealAddress_Pro:=ARDSStationZoneHeight[4].lrZone4Range,
ARrLrealAddress_Hmi:=Arm1Pos4thStage[4]);

ARfbHMIAddMappingLreal[34](
bEN:=TRUE ,
ARrLrealAddress_Pro:=ARDSStationZoneHeight[4].lrBottomPos,
ARrLrealAddress_Hmi:=Arm1BottomPos[4]);

ARfbHMIAddMappingLreal[35](
bEN:=TRUE ,
ARrLrealAddress_Pro:=ARDSStationZoneHeight[4].lrMidPos,
ARrLrealAddress_Hmi:=Arm1MidPos[4]);


(*Station 5*)

ARfbHMIAddMappingLreal[36](
bEN:=TRUE ,
ARrLrealAddress_Pro:=ARDSStationZoneHeight[5].lrTopPos,
ARrLrealAddress_Hmi:=Arm1TopPos[5]);

ARfbHMIAddMappingLreal[37](
bEN:=TRUE ,
ARrLrealAddress_Pro:=ARDSStationZoneHeight[5].lrZone1Range,
ARrLrealAddress_Hmi:=Arm1Pos1stStage[5]);

ARfbHMIAddMappingLreal[38](
bEN:=TRUE ,
ARrLrealAddress_Pro:=ARDSStationZoneHeight[5].lrZone2Range,
ARrLrealAddress_Hmi:=Arm1Pos2ndStage[5]);

ARfbHMIAddMappingLreal[39](
bEN:=TRUE ,
ARrLrealAddress_Pro:=ARDSStationZoneHeight[5].lrZone3Range,
ARrLrealAddress_Hmi:=Arm1Pos3rdStage[5]);

ARfbHMIAddMappingLreal[40](
bEN:=TRUE ,
ARrLrealAddress_Pro:=ARDSStationZoneHeight[5].lrZone4Range,
ARrLrealAddress_Hmi:=Arm1Pos4thStage[5]);

ARfbHMIAddMappingLreal[41](
bEN:=TRUE ,
ARrLrealAddress_Pro:=ARDSStationZoneHeight[5].lrBottomPos,
ARrLrealAddress_Hmi:=Arm1BottomPos[5]);

ARfbHMIAddMappingLreal[42](
bEN:=TRUE ,
ARrLrealAddress_Pro:=ARDSStationZoneHeight[5].lrMidPos,
ARrLrealAddress_Hmi:=Arm1MidPos[5]);


(*Station 6*)

ARfbHMIAddMappingLreal[43](
bEN:=TRUE ,
ARrLrealAddress_Pro:=ARDSStationZoneHeight[6].lrTopPos,
ARrLrealAddress_Hmi:=Arm1TopPos[6]);

ARfbHMIAddMappingLreal[44](
bEN:=TRUE ,
ARrLrealAddress_Pro:=ARDSStationZoneHeight[6].lrZone1Range,
ARrLrealAddress_Hmi:=Arm1Pos1stStage[6]);

ARfbHMIAddMappingLreal[45](
bEN:=TRUE ,
ARrLrealAddress_Pro:=ARDSStationZoneHeight[6].lrZone2Range,
ARrLrealAddress_Hmi:=Arm1Pos2ndStage[6]);

ARfbHMIAddMappingLreal[46](
bEN:=TRUE ,
ARrLrealAddress_Pro:=ARDSStationZoneHeight[6].lrZone3Range,
ARrLrealAddress_Hmi:=Arm1Pos3rdStage[6]);

ARfbHMIAddMappingLreal[47](
bEN:=TRUE ,
ARrLrealAddress_Pro:=ARDSStationZoneHeight[6].lrZone4Range,
ARrLrealAddress_Hmi:=Arm1Pos4thStage[6]);

ARfbHMIAddMappingLreal[48](
bEN:=TRUE ,
ARrLrealAddress_Pro:=ARDSStationZoneHeight[6].lrBottomPos,
ARrLrealAddress_Hmi:=Arm1BottomPos[6]);

ARfbHMIAddMappingLreal[49](
bEN:=TRUE ,
ARrLrealAddress_Pro:=ARDSStationZoneHeight[6].lrMidPos,
ARrLrealAddress_Hmi:=Arm1MidPos[6]);


(*Station 7*)

ARfbHMIAddMappingLreal[50](
bEN:=TRUE ,
ARrLrealAddress_Pro:=ARDSStationZoneHeight[7].lrTopPos,
ARrLrealAddress_Hmi:=Arm1TopPos[7]);

ARfbHMIAddMappingLreal[51](
bEN:=TRUE ,
ARrLrealAddress_Pro:=ARDSStationZoneHeight[7].lrZone1Range,
ARrLrealAddress_Hmi:=Arm1Pos1stStage[7]);

ARfbHMIAddMappingLreal[52](
bEN:=TRUE ,
ARrLrealAddress_Pro:=ARDSStationZoneHeight[7].lrZone2Range,
ARrLrealAddress_Hmi:=Arm1Pos2ndStage[7]);

ARfbHMIAddMappingLreal[53](
bEN:=TRUE ,
ARrLrealAddress_Pro:=ARDSStationZoneHeight[7].lrZone3Range,
ARrLrealAddress_Hmi:=Arm1Pos3rdStage[7]);

ARfbHMIAddMappingLreal[54](
bEN:=TRUE ,
ARrLrealAddress_Pro:=ARDSStationZoneHeight[7].lrZone4Range,
ARrLrealAddress_Hmi:=Arm1Pos4thStage[7]);

ARfbHMIAddMappingLreal[55](
bEN:=TRUE ,
ARrLrealAddress_Pro:=ARDSStationZoneHeight[7].lrBottomPos,
ARrLrealAddress_Hmi:=Arm1BottomPos[7]);

ARfbHMIAddMappingLreal[56](
bEN:=TRUE ,
ARrLrealAddress_Pro:=ARDSStationZoneHeight[7].lrMidPos,
ARrLrealAddress_Hmi:=Arm1MidPos[7]);


(*Station 8*)

ARfbHMIAddMappingLreal[57](
bEN:=TRUE ,
ARrLrealAddress_Pro:=ARDSStationZoneHeight[8].lrTopPos,
ARrLrealAddress_Hmi:=Arm1TopPos[8]);

ARfbHMIAddMappingLreal[58](
bEN:=TRUE ,
ARrLrealAddress_Pro:=ARDSStationZoneHeight[8].lrZone1Range,
ARrLrealAddress_Hmi:=Arm1Pos1stStage[8]);

ARfbHMIAddMappingLreal[59](
bEN:=TRUE ,
ARrLrealAddress_Pro:=ARDSStationZoneHeight[8].lrZone2Range,
ARrLrealAddress_Hmi:=Arm1Pos2ndStage[8]);

ARfbHMIAddMappingLreal[60](
bEN:=TRUE ,
ARrLrealAddress_Pro:=ARDSStationZoneHeight[8].lrZone3Range,
ARrLrealAddress_Hmi:=Arm1Pos3rdStage[8]);

ARfbHMIAddMappingLreal[61](
bEN:=TRUE ,
ARrLrealAddress_Pro:=ARDSStationZoneHeight[8].lrZone4Range,
ARrLrealAddress_Hmi:=Arm1Pos4thStage[8]);

ARfbHMIAddMappingLreal[62](
bEN:=TRUE ,
ARrLrealAddress_Pro:=ARDSStationZoneHeight[8].lrBottomPos,
ARrLrealAddress_Hmi:=Arm1BottomPos[8]);

ARfbHMIAddMappingLreal[63](
bEN:=TRUE ,
ARrLrealAddress_Pro:=ARDSStationZoneHeight[8].lrMidPos,
ARrLrealAddress_Hmi:=Arm1MidPos[8]);


(*Station 9*)

ARfbHMIAddMappingLreal[64](
bEN:=TRUE ,
ARrLrealAddress_Pro:=ARDSStationZoneHeight[9].lrTopPos,
ARrLrealAddress_Hmi:=Arm1TopPos[9]);

ARfbHMIAddMappingLreal[65](
bEN:=TRUE ,
ARrLrealAddress_Pro:=ARDSStationZoneHeight[9].lrZone1Range,
ARrLrealAddress_Hmi:=Arm1Pos1stStage[9]);

ARfbHMIAddMappingLreal[66](
bEN:=TRUE ,
ARrLrealAddress_Pro:=ARDSStationZoneHeight[9].lrZone2Range,
ARrLrealAddress_Hmi:=Arm1Pos2ndStage[9]);

ARfbHMIAddMappingLreal[67](
bEN:=TRUE ,
ARrLrealAddress_Pro:=ARDSStationZoneHeight[9].lrZone3Range,
ARrLrealAddress_Hmi:=Arm1Pos3rdStage[9]);

ARfbHMIAddMappingLreal[68](
bEN:=TRUE ,
ARrLrealAddress_Pro:=ARDSStationZoneHeight[9].lrZone4Range,
ARrLrealAddress_Hmi:=Arm1Pos4thStage[9]);

ARfbHMIAddMappingLreal[69](
bEN:=TRUE ,
ARrLrealAddress_Pro:=ARDSStationZoneHeight[9].lrBottomPos,
ARrLrealAddress_Hmi:=Arm1BottomPos[9]);

ARfbHMIAddMappingLreal[70](
bEN:=TRUE ,
ARrLrealAddress_Pro:=ARDSStationZoneHeight[9].lrMidPos,
ARrLrealAddress_Hmi:=Arm1MidPos[9]);


(*Station 10*)

ARfbHMIAddMappingLreal[71](
bEN:=TRUE ,
ARrLrealAddress_Pro:=ARDSStationZoneHeight[10].lrTopPos,
ARrLrealAddress_Hmi:=Arm1TopPos[10]);

ARfbHMIAddMappingLreal[72](
bEN:=TRUE ,
ARrLrealAddress_Pro:=ARDSStationZoneHeight[10].lrZone1Range,
ARrLrealAddress_Hmi:=Arm1Pos1stStage[10]);

ARfbHMIAddMappingLreal[73](
bEN:=TRUE ,
ARrLrealAddress_Pro:=ARDSStationZoneHeight[10].lrZone2Range,
ARrLrealAddress_Hmi:=Arm1Pos2ndStage[10]);

ARfbHMIAddMappingLreal[74](
bEN:=TRUE ,
ARrLrealAddress_Pro:=ARDSStationZoneHeight[10].lrZone3Range,
ARrLrealAddress_Hmi:=Arm1Pos3rdStage[10]);

ARfbHMIAddMappingLreal[75](
bEN:=TRUE ,
ARrLrealAddress_Pro:=ARDSStationZoneHeight[10].lrZone4Range,
ARrLrealAddress_Hmi:=Arm1Pos4thStage[10]);

ARfbHMIAddMappingLreal[76](
bEN:=TRUE ,
ARrLrealAddress_Pro:=ARDSStationZoneHeight[10].lrBottomPos,
ARrLrealAddress_Hmi:=Arm1BottomPos[10]);

ARfbHMIAddMappingLreal[77](
bEN:=TRUE ,
ARrLrealAddress_Pro:=ARDSStationZoneHeight[10].lrMidPos,
ARrLrealAddress_Hmi:=Arm1MidPos[10]);


(*Station 11*)

ARfbHMIAddMappingLreal[78](
bEN:=TRUE ,
ARrLrealAddress_Pro:=ARDSStationZoneHeight[11].lrTopPos,
ARrLrealAddress_Hmi:=Arm2TopPos[11]);

ARfbHMIAddMappingLreal[79](
bEN:=TRUE ,
ARrLrealAddress_Pro:=ARDSStationZoneHeight[11].lrZone1Range,
ARrLrealAddress_Hmi:=Arm2Pos1stStage[11]);

ARfbHMIAddMappingLreal[80](
bEN:=TRUE ,
ARrLrealAddress_Pro:=ARDSStationZoneHeight[11].lrZone2Range,
ARrLrealAddress_Hmi:=Arm2Pos2ndStage[11]);

ARfbHMIAddMappingLreal[81](
bEN:=TRUE ,
ARrLrealAddress_Pro:=ARDSStationZoneHeight[11].lrZone3Range,
ARrLrealAddress_Hmi:=Arm2Pos3rdStage[11]);

ARfbHMIAddMappingLreal[82](
bEN:=TRUE ,
ARrLrealAddress_Pro:=ARDSStationZoneHeight[11].lrZone4Range,
ARrLrealAddress_Hmi:=Arm2Pos4thStage[11]);

ARfbHMIAddMappingLreal[83](
bEN:=TRUE ,
ARrLrealAddress_Pro:=ARDSStationZoneHeight[11].lrBottomPos,
ARrLrealAddress_Hmi:=Arm2BottomPos[11]);

ARfbHMIAddMappingLreal[84](
bEN:=TRUE ,
ARrLrealAddress_Pro:=ARDSStationZoneHeight[11].lrMidPos,
ARrLrealAddress_Hmi:=Arm2MidPos[11]);


(*Station 12*)

ARfbHMIAddMappingLreal[85](
bEN:=TRUE ,
ARrLrealAddress_Pro:=ARDSStationZoneHeight[12].lrTopPos,
ARrLrealAddress_Hmi:=Arm2TopPos[12]);

ARfbHMIAddMappingLreal[86](
bEN:=TRUE ,
ARrLrealAddress_Pro:=ARDSStationZoneHeight[12].lrZone1Range,
ARrLrealAddress_Hmi:=Arm2Pos1stStage[12]);

ARfbHMIAddMappingLreal[87](
bEN:=TRUE ,
ARrLrealAddress_Pro:=ARDSStationZoneHeight[12].lrZone2Range,
ARrLrealAddress_Hmi:=Arm2Pos2ndStage[12]);

ARfbHMIAddMappingLreal[88](
bEN:=TRUE ,
ARrLrealAddress_Pro:=ARDSStationZoneHeight[12].lrZone3Range,
ARrLrealAddress_Hmi:=Arm2Pos3rdStage[12]);

ARfbHMIAddMappingLreal[89](
bEN:=TRUE ,
ARrLrealAddress_Pro:=ARDSStationZoneHeight[12].lrZone4Range,
ARrLrealAddress_Hmi:=Arm2Pos4thStage[12]);

ARfbHMIAddMappingLreal[90](
bEN:=TRUE ,
ARrLrealAddress_Pro:=ARDSStationZoneHeight[12].lrBottomPos,
ARrLrealAddress_Hmi:=Arm2BottomPos[12]);

ARfbHMIAddMappingLreal[91](
bEN:=TRUE ,
ARrLrealAddress_Pro:=ARDSStationZoneHeight[12].lrMidPos,
ARrLrealAddress_Hmi:=Arm2MidPos[12]);


(*Unloading*)

ARfbHMIAddMappingLreal[92](
bEN:=TRUE ,
ARrLrealAddress_Pro:=ARDSUldZoneHeight[1].lrTopPos,
ARrLrealAddress_Hmi:=Arm1TopPos[20]);

ARfbHMIAddMappingLreal[93](
bEN:=TRUE ,
ARrLrealAddress_Pro:=ARDSUldZoneHeight[1].lrZone1Range,
ARrLrealAddress_Hmi:=Arm1Pos1stStage[20]);

ARfbHMIAddMappingLreal[94](
bEN:=TRUE ,
ARrLrealAddress_Pro:=ARDSUldZoneHeight[1].lrZone2Range,
ARrLrealAddress_Hmi:=Arm1Pos2ndStage[20]);

ARfbHMIAddMappingLreal[95](
bEN:=TRUE ,
ARrLrealAddress_Pro:=ARDSUldZoneHeight[1].lrZone3Range,
ARrLrealAddress_Hmi:=Arm1Pos3rdStage[20]);

ARfbHMIAddMappingLreal[96](
bEN:=TRUE ,
ARrLrealAddress_Pro:=ARDSUldZoneHeight[1].lrZone4Range,
ARrLrealAddress_Hmi:=Arm1Pos4thStage[20]);

ARfbHMIAddMappingLreal[97](
bEN:=TRUE ,
ARrLrealAddress_Pro:=ARDSUldZoneHeight[1].lrBottomPos,
ARrLrealAddress_Hmi:=Arm1BottomPos[20]);

ARfbHMIAddMappingLreal[98](
bEN:=TRUE ,
ARrLrealAddress_Pro:=ARDSUldZoneHeight[1].lrMidPos,
ARrLrealAddress_Hmi:=Arm1MidPos[20]);



IF mb_Output_Registers[39] > 0 THEN
	ARfbHMIAddMappingReal_Word[39](
		bEN:= TRUE ,
		ARrRealAddress_Pro:= ARrStnTempSV[1],
		ARwAddress_Hmi:= mb_Output_Registers[39]);
END_IF

IF mb_Output_Registers[40] > 0 THEN
	ARfbHMIAddMappingReal_Word[40](
		bEN:= TRUE ,
		ARrRealAddress_Pro:= ARrStnTempSV[2],
		ARwAddress_Hmi:= mb_Output_Registers[40]);
END_IF

IF mb_Output_Registers[41] > 0 THEN
	ARfbHMIAddMappingReal_Word[41](
		bEN:= TRUE ,
		ARrRealAddress_Pro:= ARrStnTempSV[3],
		ARwAddress_Hmi:= mb_Output_Registers[41]);
END_IF

IF mb_Output_Registers[42] > 0 THEN
	ARfbHMIAddMappingReal_Word[42](
		bEN:= TRUE ,
		ARrRealAddress_Pro:= ARrStnTempSV[4],
		ARwAddress_Hmi:= mb_Output_Registers[42]);
END_IF

IF mb_Output_Registers[43] > 0 THEN
	ARfbHMIAddMappingReal_Word[43](
		bEN:= TRUE ,
		ARrRealAddress_Pro:= ARrStnTempSV[5],
		ARwAddress_Hmi:= mb_Output_Registers[43]);
END_IF

IF mb_Output_Registers[44] > 0 THEN
	ARfbHMIAddMappingReal_Word[44](
		bEN:= TRUE ,
		ARrRealAddress_Pro:= ARrStnTempSV[6],
		ARwAddress_Hmi:= mb_Output_Registers[44]);
END_IF

IF mb_Output_Registers[45] > 0 THEN
	ARfbHMIAddMappingReal_Word[45](
		bEN:= TRUE ,
		ARrRealAddress_Pro:= ARrStnTempSV[7],
		ARwAddress_Hmi:= mb_Output_Registers[45]);
END_IF

END_PROGRAM

// ---- FBs/B_JKS_NewFB/FBP-HMIAddMapping/fbHMIAddMappingLreal.TcPOU
FUNCTION_BLOCK fbHMIAddMappingLreal


VAR_INPUT
	bEN : BOOL;
END_VAR

VAR_IN_OUT PERSISTENT
	ARrLrealAddress_Pro 					: LREAL;
	ARrLrealAddress_Hmi 				: LREAL;
END_VAR


VAR_OUTPUT
END_VAR


VAR
	ARBufferrLrealAddress_Pro 				:  LREAL;
	ARBufferrLrealAddress_Hmi 				:  LREAL;

	ARUpdate_bLrealAddress_Pro 				:  BOOL;
	ARUpdate_bLrealAddress_Hmi 				:  BOOL;

END_VAR
VAR
	bENRE : R_TRIG;

	ProSideFL: LREAL;
	HmiSideFL: LREAL;
END_VAR

(*Initialized*)
bENRE(CLK:=bEN , Q=> );
IF bENRE.Q THEN
			(*Int*)
			ARBufferrLrealAddress_Pro := ARrLrealAddress_Pro;
			ARBufferrLrealAddress_Hmi := ARrLrealAddress_Pro;
			ARrLrealAddress_Hmi := ARrLrealAddress_Pro;
END_IF

(*Program*)


ARUpdate_bLrealAddress_Pro := FALSE;

	IF ARBufferrLrealAddress_Pro <> ARrLrealAddress_Pro THEN
		ARUpdate_bLrealAddress_Pro := TRUE;
	END_IF

	IF ARUpdate_bLrealAddress_Pro THEN
		ARBufferrLrealAddress_Pro := ARrLrealAddress_Pro;
		ARBufferrLrealAddress_Hmi := ARrLrealAddress_Pro;
		ARrLrealAddress_Hmi := ARrLrealAddress_Pro;
	END_IF



			(**********HMI Side Value Change**********)

ARUpdate_bLrealAddress_Hmi := FALSE;

	(**********Int**********)
	IF ARBufferrLrealAddress_Hmi <> ARrLrealAddress_Hmi THEN
		ARUpdate_bLrealAddress_Hmi := TRUE;
	END_IF

	IF ARUpdate_bLrealAddress_Hmi THEN
		ARBufferrLrealAddress_Pro := ARrLrealAddress_Hmi;
		ARBufferrLrealAddress_Hmi := ARrLrealAddress_Hmi;
		ARrLrealAddress_Pro := ARrLrealAddress_Hmi;
	END_IF

END_FUNCTION_BLOCK

// ---- FBs/B_JKS_NewFB/FBP-HMIAddMapping/fbHMIAddMappingInt_Word.TcPOU
FUNCTION_BLOCK fbHMIAddMappingInt_Word


VAR_INPUT
	bEN : BOOL;
END_VAR

VAR_IN_OUT PERSISTENT
	ARiIntAddress_Pro 					: INT;
	ARwAddress_Hmi 					: WORD;
END_VAR


VAR_OUTPUT
END_VAR


VAR
	ARBufferiIntAddress_Pro 					:  INT;
	ARBufferwAddress_Hmi 					:  WORD;

	ARUpdate_bIntAddress_Pro 				:  BOOL;
	ARUpdate_bWordAddress_Hmi 			:  BOOL;

END_VAR
VAR
	bENRE : R_TRIG;

	ProSideFL: REAL;
	HmiSideFL: REAL;
END_VAR

(*Initialized*)
bENRE(CLK:=bEN , Q=> );
IF bENRE.Q THEN
			(*Int*)
			ARBufferiIntAddress_Pro := ARiIntAddress_Pro;
			ARBufferwAddress_Hmi := INT_TO_WORD(ARiIntAddress_Pro);
			ARwAddress_Hmi := INT_TO_WORD(ARiIntAddress_Pro);
END_IF

(*Program*)


ARUpdate_bIntAddress_Pro := FALSE;

	IF ARBufferiIntAddress_Pro <> ARiIntAddress_Pro THEN
		ARUpdate_bIntAddress_Pro := TRUE;
	END_IF

	IF ARUpdate_bIntAddress_Pro THEN
		ARBufferiIntAddress_Pro := ARiIntAddress_Pro;
		ARBufferwAddress_Hmi := INT_TO_WORD(ARiIntAddress_Pro);
		ARwAddress_Hmi := INT_TO_WORD(ARiIntAddress_Pro);
	END_IF



			(**********HMI Side Value Change**********)

ARUpdate_bWordAddress_Hmi := FALSE;

	(**********Int**********)
	IF ARBufferwAddress_Hmi <> ARwAddress_Hmi THEN
		ARUpdate_bWordAddress_Hmi := TRUE;
	END_IF

	IF ARUpdate_bWordAddress_Hmi THEN
		ARBufferiIntAddress_Pro := WORD_TO_INT(ARwAddress_Hmi);
		ARBufferwAddress_Hmi := ARwAddress_Hmi;
		ARiIntAddress_Pro := WORD_TO_INT(ARwAddress_Hmi);
	END_IF

END_FUNCTION_BLOCK

// ---- FBs/B_JKS_NewFB/FBP-HMIAddMapping/fbHMIAddMappingReal_Word.TcPOU
FUNCTION_BLOCK fbHMIAddMappingReal_Word


VAR_INPUT
	bEN : BOOL;
END_VAR

VAR_IN_OUT PERSISTENT
	ARrRealAddress_Pro 					: REAL;
	ARwAddress_Hmi 					: WORD;
END_VAR


VAR_OUTPUT
END_VAR


VAR
	ARBufferrRealAddress_Pro 				:  REAL;
	ARBufferwAddress_Hmi 					:  WORD;

	ARUpdate_bRealAddress_Pro 				:  BOOL;
	ARUpdate_bWordAddress_Hmi 			:  BOOL;

END_VAR
VAR
	bENRE : R_TRIG;

	ProSideFL: REAL;
	HmiSideFL: REAL;
END_VAR

(*Initialized*)
bENRE(CLK:=bEN , Q=> );
IF bENRE.Q THEN
			(*Int*)
			ARBufferrRealAddress_Pro := ARrRealAddress_Pro;
			ARBufferwAddress_Hmi := REAL_TO_WORD(ARrRealAddress_Pro);
			ARwAddress_Hmi := REAL_TO_WORD(ARrRealAddress_Pro);
END_IF

(*Program*)


ARUpdate_bRealAddress_Pro := FALSE;

	IF ARBufferrRealAddress_Pro <> ARrRealAddress_Pro THEN
		ARUpdate_bRealAddress_Pro := TRUE;
	END_IF

	IF ARUpdate_bRealAddress_Pro THEN
		ARBufferrRealAddress_Pro := ARrRealAddress_Pro;
		ARBufferwAddress_Hmi := REAL_TO_WORD(ARrRealAddress_Pro);
		ARwAddress_Hmi := REAL_TO_WORD(ARrRealAddress_Pro);
	END_IF



			(**********HMI Side Value Change**********)

ARUpdate_bWordAddress_Hmi := FALSE;

	(**********Int**********)
	IF ARBufferwAddress_Hmi <> ARwAddress_Hmi THEN
		ARUpdate_bWordAddress_Hmi := TRUE;
	END_IF

	IF ARUpdate_bWordAddress_Hmi THEN
		ARBufferrRealAddress_Pro := WORD_TO_REAL(ARwAddress_Hmi);
		ARBufferwAddress_Hmi := ARwAddress_Hmi;
		ARrRealAddress_Pro := WORD_TO_REAL(ARwAddress_Hmi);
	END_IF

END_FUNCTION_BLOCK

// ---- POUs/MainProgram/Other/HMI_Function.TcPOU
PROGRAM HMI_Function
VAR


	(*fbDetergentPBresetPassword:fbDetergent_BasketQuantityResetPB_PasswordControl;*)

	iRecipeNoFeed:INT;

	MotionX :LREAL;
	MotionY:LREAL;

	MotionX_1 :LREAL;
	MotionY_1:LREAL;

	sProductRecipeStepSeqRecipeDescription : ARRAY [1..20] OF STRING(99);
	ARsUpPickPatternDescription: ARRAY [1..20] OF STRING(99);
	ARsDownTransferPatternDescription : ARRAY [1..20] OF STRING(99);

(*Recipe Barcode Page Description*)

	iRegNoM				:INT;

END_VAR

(*Recipe Description*)
sProductRecipeStepSeqRecipeDescription[1]:=sProductRecipeStep1SeqRecipeDescription;
sProductRecipeStepSeqRecipeDescription[2]:=sProductRecipeStep2SeqRecipeDescription;
sProductRecipeStepSeqRecipeDescription[3]:=sProductRecipeStep3SeqRecipeDescription;
sProductRecipeStepSeqRecipeDescription[4]:=sProductRecipeStep4SeqRecipeDescription;
sProductRecipeStepSeqRecipeDescription[5]:=sProductRecipeStep5SeqRecipeDescription;
sProductRecipeStepSeqRecipeDescription[6]:=sProductRecipeStep6SeqRecipeDescription;
sProductRecipeStepSeqRecipeDescription[7]:=sProductRecipeStep7SeqRecipeDescription;
sProductRecipeStepSeqRecipeDescription[8]:=sProductRecipeStep8SeqRecipeDescription;
sProductRecipeStepSeqRecipeDescription[9]:=sProductRecipeStep9SeqRecipeDescription;
sProductRecipeStepSeqRecipeDescription[10]:=sProductRecipeStep10SeqRecipeDescription;
sProductRecipeStepSeqRecipeDescription[11]:=sProductRecipeStep11SeqRecipeDescription;
sProductRecipeStepSeqRecipeDescription[12]:=sProductRecipeStep12SeqRecipeDescription;
sProductRecipeStepSeqRecipeDescription[13]:=sProductRecipeStep13SeqRecipeDescription;
sProductRecipeStepSeqRecipeDescription[14]:=sProductRecipeStep14SeqRecipeDescription;
sProductRecipeStepSeqRecipeDescription[15]:=sProductRecipeStep15SeqRecipeDescription;
sProductRecipeStepSeqRecipeDescription[16]:=sProductRecipeStep16SeqRecipeDescription;
sProductRecipeStepSeqRecipeDescription[17]:=sProductRecipeStep17SeqRecipeDescription;
sProductRecipeStepSeqRecipeDescription[18]:=sProductRecipeStep18SeqRecipeDescription;
sProductRecipeStepSeqRecipeDescription[19]:=sProductRecipeStep19SeqRecipeDescription;
sProductRecipeStepSeqRecipeDescription[20]:=sProductRecipeStep20SeqRecipeDescription;

(*Up transfer Description*)

ARsUpPickPatternDescription[1]:=ARsUpPickPatternDescription1;
ARsUpPickPatternDescription[2]:=ARsUpPickPatternDescription2;
ARsUpPickPatternDescription[3]:=ARsUpPickPatternDescription3;
ARsUpPickPatternDescription[4]:=ARsUpPickPatternDescription4;
ARsUpPickPatternDescription[5]:=ARsUpPickPatternDescription5;
ARsUpPickPatternDescription[6]:=ARsUpPickPatternDescription6;
ARsUpPickPatternDescription[7]:=ARsUpPickPatternDescription7;
ARsUpPickPatternDescription[8]:=ARsUpPickPatternDescription8;
ARsUpPickPatternDescription[9]:=ARsUpPickPatternDescription9;
ARsUpPickPatternDescription[10]:=ARsUpPickPatternDescription10;
ARsUpPickPatternDescription[11]:=ARsUpPickPatternDescription11;
ARsUpPickPatternDescription[12]:=ARsUpPickPatternDescription12;
ARsUpPickPatternDescription[13]:=ARsUpPickPatternDescription13;
ARsUpPickPatternDescription[14]:=ARsUpPickPatternDescription14;
ARsUpPickPatternDescription[15]:=ARsUpPickPatternDescription15;
ARsUpPickPatternDescription[16]:=ARsUpPickPatternDescription16;
ARsUpPickPatternDescription[17]:=ARsUpPickPatternDescription17;
ARsUpPickPatternDescription[18]:=ARsUpPickPatternDescription18;
ARsUpPickPatternDescription[19]:=ARsUpPickPatternDescription19;
ARsUpPickPatternDescription[20]:=ARsUpPickPatternDescription20;

(*Down transfer Description*)


ARsDownTransferPatternDescription[1]:=ARsDownTransferPatternDescription1;
ARsDownTransferPatternDescription[2]:=ARsDownTransferPatternDescription2;
ARsDownTransferPatternDescription[3]:=ARsDownTransferPatternDescription3;
ARsDownTransferPatternDescription[4]:=ARsDownTransferPatternDescription4;
ARsDownTransferPatternDescription[5]:=ARsDownTransferPatternDescription5;
ARsDownTransferPatternDescription[6]:=ARsDownTransferPatternDescription6;
ARsDownTransferPatternDescription[7]:=ARsDownTransferPatternDescription7;
ARsDownTransferPatternDescription[8]:=ARsDownTransferPatternDescription8;
ARsDownTransferPatternDescription[9]:=ARsDownTransferPatternDescription9;
ARsDownTransferPatternDescription[10]:=ARsDownTransferPatternDescription10;
ARsDownTransferPatternDescription[11]:=ARsDownTransferPatternDescription11;
ARsDownTransferPatternDescription[12]:=ARsDownTransferPatternDescription12;
ARsDownTransferPatternDescription[13]:=ARsDownTransferPatternDescription13;
ARsDownTransferPatternDescription[14]:=ARsDownTransferPatternDescription14;
ARsDownTransferPatternDescription[15]:=ARsDownTransferPatternDescription15;
ARsDownTransferPatternDescription[16]:=ARsDownTransferPatternDescription16;
ARsDownTransferPatternDescription[17]:=ARsDownTransferPatternDescription17;
ARsDownTransferPatternDescription[18]:=ARsDownTransferPatternDescription18;
ARsDownTransferPatternDescription[19]:=ARsDownTransferPatternDescription19;
ARsDownTransferPatternDescription[20]:=ARsDownTransferPatternDescription20;

	(*Tracker No Array Set*)



TrackeriArrayNo[1]:=TimeTrackerPage+1;
TrackeriArrayNo[2]:=TimeTrackerPage+2;
TrackeriArrayNo[3]:=TimeTrackerPage+3;
TrackeriArrayNo[4]:=TimeTrackerPage+4;
TrackeriArrayNo[5]:=TimeTrackerPage+5;
TrackeriArrayNo[6]:=TimeTrackerPage+6;
TrackeriArrayNo[7]:=TimeTrackerPage+7;
TrackeriArrayNo[8]:=TimeTrackerPage+8;
TrackeriArrayNo[9]:=TimeTrackerPage+9;
TrackeriArrayNo[10]:=TimeTrackerPage+10;
TrackeriArrayNo[11]:=TimeTrackerPage+11;
TrackeriArrayNo[12]:=TimeTrackerPage+12;
TrackeriArrayNo[13]:=TimeTrackerPage+13;
TrackeriArrayNo[14]:=TimeTrackerPage+14;
TrackeriArrayNo[15]:=TimeTrackerPage+15;
TrackeriArrayNo[16]:=TimeTrackerPage+16;
TrackeriArrayNo[17]:=TimeTrackerPage+17;
TrackeriArrayNo[18]:=TimeTrackerPage+18;
TrackeriArrayNo[19]:=TimeTrackerPage+19;
TrackeriArrayNo[20]:=TimeTrackerPage+20;

	(*Recipe Descripin for recipe Editor page*)

sRecipeDescriptionStep[1]:=sProductRecipeStep1SeqRecipeDescription;
sRecipeDescriptionStep[2]:=sProductRecipeStep2SeqRecipeDescription;
sRecipeDescriptionStep[3]:=sProductRecipeStep3SeqRecipeDescription;
sRecipeDescriptionStep[4]:=sProductRecipeStep4SeqRecipeDescription;
sRecipeDescriptionStep[5]:=sProductRecipeStep5SeqRecipeDescription;
sRecipeDescriptionStep[6]:=sProductRecipeStep6SeqRecipeDescription;
sRecipeDescriptionStep[7]:=sProductRecipeStep7SeqRecipeDescription;
sRecipeDescriptionStep[8]:=sProductRecipeStep8SeqRecipeDescription;
sRecipeDescriptionStep[9]:=sProductRecipeStep9SeqRecipeDescription;
sRecipeDescriptionStep[10]:=sProductRecipeStep10SeqRecipeDescription;

sRecipeDescriptionStep[11]:=sProductRecipeStep11SeqRecipeDescription;
sRecipeDescriptionStep[12]:=sProductRecipeStep12SeqRecipeDescription;
sRecipeDescriptionStep[13]:=sProductRecipeStep13SeqRecipeDescription;
sRecipeDescriptionStep[14]:=sProductRecipeStep14SeqRecipeDescription;
sRecipeDescriptionStep[15]:=sProductRecipeStep15SeqRecipeDescription;
sRecipeDescriptionStep[16]:=sProductRecipeStep16SeqRecipeDescription;
sRecipeDescriptionStep[17]:=sProductRecipeStep17SeqRecipeDescription;
sRecipeDescriptionStep[18]:=sProductRecipeStep18SeqRecipeDescription;
sRecipeDescriptionStep[19]:=sProductRecipeStep19SeqRecipeDescription;
sRecipeDescriptionStep[20]:=sProductRecipeStep20SeqRecipeDescription;

(*iCurrentScreenNo:= iAutoInfoNo;*)
iCurrentScreenNo:= iStationNo;

(*7Days Remap*)

ArbDayOnEn_IN[1]:=Day1En[1];
ArbDayOnEn_IN[2]:=Day2En[1];
ArbDayOnEn_IN[3]:=Day3En[1];
ArbDayOnEn_IN[4]:=Day4En[1];
ArbDayOnEn_IN[5]:=Day5En[1];
ArbDayOnEn_IN[6]:=Day6En[1];
ArbDayOnEn_IN[7]:=Day7En[1];

ArbDayOffEn_IN[1]:=Day1En[2];
ArbDayOffEn_IN[2]:=Day2En[2];
ArbDayOffEn_IN[3]:=Day3En[2];
ArbDayOffEn_IN[4]:=Day4En[2];
ArbDayOffEn_IN[5]:=Day5En[2];
ArbDayOffEn_IN[6]:=Day6En[2];
ArbDayOffEn_IN[7]:=Day7En[2];


ArwDayOnHour_IN[1]:=Day1H[1];
ArwDayOnHour_IN[2]:=Day2H[1];
ArwDayOnHour_IN[3]:=Day3H[1];
ArwDayOnHour_IN[4]:=Day4H[1];
ArwDayOnHour_IN[5]:=Day5H[1];
ArwDayOnHour_IN[6]:=Day6H[1];
ArwDayOnHour_IN[7]:=Day7H[1];

ArwDayOffHour_IN[1]:=Day1H[2];
ArwDayOffHour_IN[2]:=Day2H[2];
ArwDayOffHour_IN[3]:=Day3H[2];
ArwDayOffHour_IN[4]:=Day4H[2];
ArwDayOffHour_IN[5]:=Day5H[2];
ArwDayOffHour_IN[6]:=Day6H[2];
ArwDayOffHour_IN[7]:=Day7H[2];


ArwDayOnMinute_IN[1]:=Day1M[1];
ArwDayOnMinute_IN[2]:=Day2M[1];
ArwDayOnMinute_IN[3]:=Day3M[1];
ArwDayOnMinute_IN[4]:=Day4M[1];
ArwDayOnMinute_IN[5]:=Day5M[1];
ArwDayOnMinute_IN[6]:=Day6M[1];
ArwDayOnMinute_IN[7]:=Day7M[1];

ArwDayOffMinute_IN[1]:=Day1M[2];
ArwDayOffMinute_IN[2]:=Day2M[2];
ArwDayOffMinute_IN[3]:=Day3M[2];
ArwDayOffMinute_IN[4]:=Day4M[2];
ArwDayOffMinute_IN[5]:=Day5M[2];
ArwDayOffMinute_IN[6]:=Day6M[2];
ArwDayOffMinute_IN[7]:=Day7M[2];


(*iArmVertCurrentPos:=LREAL_TO_INT(ARlrVertPositionMM[1]/lrVertHmiRatio);*)
xRatio(*:=11*);
YRatio;

xRatio_1;
yRatio_1:=20;

IF  ARbArmVertHomeDone[1] AND ARbArmHorzHomeDone[1] THEN
bArmHomingComplete[1]:=TRUE;
ELSE
bArmHomingComplete[1]:=FALSE;
END_IF

IF ARbArmVertHomeDone[2] AND ARbArmHorzHomeDone[2] THEN
bArmHomingComplete[2]:=TRUE;
ELSE
bArmHomingComplete[2]:=FALSE;
END_IF


IF DSArm1HorzConfig.lrGen_Out_CurrentPos (*ARlrHorzPositionMM[1]*)>0 AND (xRatio <> 0) THEN
	MotionX:=(DSArm1HorzConfig.lrGen_Out_CurrentPos (*ARlrHorzPositionMM[1]*)/xRatio);
END_IF

IF DSArm1VertConfig.lrGen_Out_CurrentPos (*ARlrVertPositionMM[1]*)>0 AND (yRatio <> 0) THEN
	MotionY:=DSArm1VertConfig.lrGen_Out_CurrentPos (*ARlrVertPositionMM[1]*)/yRatio;
END_IF


IF DSArm2HorzConfig.lrGen_Out_CurrentPos (*ARlrHorzPositionMM[2]*)>0 AND (xRatio_1 <> 0) THEN
	MotionX_1:=DSArm2HorzConfig.lrGen_Out_CurrentPos (*ARlrHorzPositionMM[2]*)/xRatio_1;
END_IF

IF DSArm2VertConfig.lrGen_Out_CurrentPos (*ARlrVertPositionMM[2]*)>0 AND (yRatio_1 <> 0) THEN
	MotionY_1:=DSArm2VertConfig.lrGen_Out_CurrentPos (*ARlrVertPositionMM[2]*)/yRatio_1;
END_IF

(*fbDetergentPBresetPassword(
	UserPassword:=UserPassword,
	ARiManualDetergentResetPassword:=ARiManualDetergentResetPassword,
	ARbManualDetergentResetFlag=>ARbManualDetergentResetFlag,);*)


(*Barcode Recipe Description*)

IF iRegNoM<30 THEN
	 iRegNoM:= iRegNoM+1;
ELSIF  iRegNoM>=30 THEN
	 iRegNoM:=0;
END_IF



IF DsAr1sG_BarcodeRegSectionDisplayHMI[iRegNoM].iLinkProductRecipeNo=1 THEN
	DsAr1sG_BarcodeRegSectionDisplayHMI[iRegNoM].sLinkProductRecipeDescription:= ARsProductRecipeDescription[1];
ELSIF DsAr1sG_BarcodeRegSectionDisplayHMI[iRegNoM].iLinkProductRecipeNo=2 THEN
	DsAr1sG_BarcodeRegSectionDisplayHMI[iRegNoM].sLinkProductRecipeDescription:= ARsProductRecipeDescription[2];
ELSIF DsAr1sG_BarcodeRegSectionDisplayHMI[iRegNoM].iLinkProductRecipeNo=3 THEN
	DsAr1sG_BarcodeRegSectionDisplayHMI[iRegNoM].sLinkProductRecipeDescription:= ARsProductRecipeDescription[3];
ELSIF DsAr1sG_BarcodeRegSectionDisplayHMI[iRegNoM].iLinkProductRecipeNo=4 THEN
	DsAr1sG_BarcodeRegSectionDisplayHMI[iRegNoM].sLinkProductRecipeDescription:= ARsProductRecipeDescription[4];
ELSIF DsAr1sG_BarcodeRegSectionDisplayHMI[iRegNoM].iLinkProductRecipeNo=5 THEN
	DsAr1sG_BarcodeRegSectionDisplayHMI[iRegNoM].sLinkProductRecipeDescription:= ARsProductRecipeDescription[5];
ELSIF DsAr1sG_BarcodeRegSectionDisplayHMI[iRegNoM].iLinkProductRecipeNo=6 THEN
	DsAr1sG_BarcodeRegSectionDisplayHMI[iRegNoM].sLinkProductRecipeDescription:= ARsProductRecipeDescription[6];
ELSIF DsAr1sG_BarcodeRegSectionDisplayHMI[iRegNoM].iLinkProductRecipeNo=7 THEN
	DsAr1sG_BarcodeRegSectionDisplayHMI[iRegNoM].sLinkProductRecipeDescription:= ARsProductRecipeDescription[7];
ELSIF DsAr1sG_BarcodeRegSectionDisplayHMI[iRegNoM].iLinkProductRecipeNo=8 THEN
	DsAr1sG_BarcodeRegSectionDisplayHMI[iRegNoM].sLinkProductRecipeDescription:= ARsProductRecipeDescription[8];
ELSIF DsAr1sG_BarcodeRegSectionDisplayHMI[iRegNoM].iLinkProductRecipeNo=9 THEN
	DsAr1sG_BarcodeRegSectionDisplayHMI[iRegNoM].sLinkProductRecipeDescription:= ARsProductRecipeDescription[9];
ELSIF DsAr1sG_BarcodeRegSectionDisplayHMI[iRegNoM].iLinkProductRecipeNo=10 THEN
	DsAr1sG_BarcodeRegSectionDisplayHMI[iRegNoM].sLinkProductRecipeDescription:= ARsProductRecipeDescription[10];
ELSIF DsAr1sG_BarcodeRegSectionDisplayHMI[iRegNoM].iLinkProductRecipeNo=11 THEN
	DsAr1sG_BarcodeRegSectionDisplayHMI[iRegNoM].sLinkProductRecipeDescription:= ARsProductRecipeDescription[11];
ELSIF DsAr1sG_BarcodeRegSectionDisplayHMI[iRegNoM].iLinkProductRecipeNo=12 THEN
	DsAr1sG_BarcodeRegSectionDisplayHMI[iRegNoM].sLinkProductRecipeDescription:= ARsProductRecipeDescription[12];
ELSIF DsAr1sG_BarcodeRegSectionDisplayHMI[iRegNoM].iLinkProductRecipeNo=13 THEN
	DsAr1sG_BarcodeRegSectionDisplayHMI[iRegNoM].sLinkProductRecipeDescription:= ARsProductRecipeDescription[13];
ELSIF DsAr1sG_BarcodeRegSectionDisplayHMI[iRegNoM].iLinkProductRecipeNo=14 THEN
	DsAr1sG_BarcodeRegSectionDisplayHMI[iRegNoM].sLinkProductRecipeDescription:= ARsProductRecipeDescription[14];
ELSIF DsAr1sG_BarcodeRegSectionDisplayHMI[iRegNoM].iLinkProductRecipeNo=15 THEN
	DsAr1sG_BarcodeRegSectionDisplayHMI[iRegNoM].sLinkProductRecipeDescription:= ARsProductRecipeDescription[15];
ELSIF DsAr1sG_BarcodeRegSectionDisplayHMI[iRegNoM].iLinkProductRecipeNo=16 THEN
	DsAr1sG_BarcodeRegSectionDisplayHMI[iRegNoM].sLinkProductRecipeDescription:= ARsProductRecipeDescription[16];
ELSIF DsAr1sG_BarcodeRegSectionDisplayHMI[iRegNoM].iLinkProductRecipeNo=17 THEN
	DsAr1sG_BarcodeRegSectionDisplayHMI[iRegNoM].sLinkProductRecipeDescription:= ARsProductRecipeDescription[17];
ELSIF DsAr1sG_BarcodeRegSectionDisplayHMI[iRegNoM].iLinkProductRecipeNo=18 THEN
	DsAr1sG_BarcodeRegSectionDisplayHMI[iRegNoM].sLinkProductRecipeDescription:= ARsProductRecipeDescription[18];
ELSIF DsAr1sG_BarcodeRegSectionDisplayHMI[iRegNoM].iLinkProductRecipeNo=19 THEN
	DsAr1sG_BarcodeRegSectionDisplayHMI[iRegNoM].sLinkProductRecipeDescription:= ARsProductRecipeDescription[19];
ELSIF DsAr1sG_BarcodeRegSectionDisplayHMI[iRegNoM].iLinkProductRecipeNo=20THEN
	DsAr1sG_BarcodeRegSectionDisplayHMI[iRegNoM].sLinkProductRecipeDescription:= ARsProductRecipeDescription[20];
ELSIF DsAr1sG_BarcodeRegSectionDisplayHMI[iRegNoM].iLinkProductRecipeNo=0 THEN
	DsAr1sG_BarcodeRegSectionDisplayHMI[iRegNoM].sLinkProductRecipeDescription:= '';
END_IF



(*Map the  Recipe Description to AR2sDSCv_LdConfirmBasketInfo[1,1].sProgramDescription during barcode Bypass Function*)

IF NOT bBarcodeBypass AND  iSecs_Control_State<>5 THEN
	iRecipeNoFeed:=iBarcodeRecipeNo_OUT;
ELSIF bBarcodeBypass AND iSecs_Control_State<>5 THEN
	iRecipeNoFeed:=iUserDefineProductRecipeNo;
ELSIF iSecs_Control_State=5 THEN
	iRecipeNoFeed:=iServerSecsGemProgNo;
END_IF

(*Map The Recipe desc to the Produc desc at Loading*)

IF AR2sDSCv_LdConfirmBasketInfo[1,1].bAvailibility THEN
	IF iRecipeNoFeed<>0 THEN
		AR2sDSCv_LdConfirmBasketInfo[1,1].sProgramDescription:=ARsProductRecipeDescription[iRecipeNoFeed];
	END_IF
END_IF

END_PROGRAM

// ---- POUs/MainProgram/Other/HoldingBit_DoorTransfer.TcPOU
PROGRAM HoldingBit_DoorTransfer
VAR

	ARfbStnDoorCtrl		: ARRAY [1..iStnQty] OF fbSlidingDoorCtrl;
	ARfbStnDoorOpen		: ARRAY [1..iStnQty] OF CMP_OC_W1;
	ARfbStnDoorClose	: ARRAY [1..iStnQty] OF CMP_OC_W1;
	
	ARfbUldDoorCtrl		:  fbSlidingDoorCtrl;
	ARfbUldDoorOpen		:  CMP_OC_W1;
	ARfbUldDoorClose	:  CMP_OC_W1;
	
	ARfbUldConveyorCtrl		:  fbSlidingDoorCtrl;
	ARfbUldConveyorOpen		:  CMP_OC_W1;
	ARfbUldConveyorClose	:  CMP_OC_W1;
	
	

	LdDoorCtrl: fbSlidingDoorCtrl;
	LdDoorOpen: CMP_OC_W1;
	LdDoorClose: CMP_OC_W1;

	UldDoorCtrl: fbSlidingDoorCtrl;
	UldDoorOpen: CMP_OC_W1;
	UldDoorClose: CMP_OC_W1;

	bArm1TransferToStn1: BOOL;
	bArm1TransferToStn2: BOOL;
	bArm1TransferToStn3 : BOOL;
	bArm1TransferToStn4 : BOOL;
	bArm1TransferToStn5 : BOOL;
	bArm1TransferToStn6: BOOL;
	bArm1TransferToStn7: BOOL;
	bArm1TransferToStn8 : BOOL;
	bArm1TransferToStn9 : BOOL;
	bArm1TransferToStn10 : BOOL;
	bArm1TransferToStn11 : BOOL;
	bArm1TransferToStn12 : BOOL;
	bArm1TransferToUld1: BOOL;

	bArm2TransferToStn8 : BOOL;
	bArm2TransferToStn9 : BOOL;
	bArm2TransferToStn10 : BOOL;
	bArm2TransferToStn11 : BOOL;

	bArmPnpStep6: BOOL;

	TON1: TON;
	TON2: TON;
	TON3: TON;
	TON4: TON;
	TON5: TON;
	TON6: TON;
	TON7: TON;
	TON8: TON;
	TON9: TON;
	TON10: TON;
	TON11: TON;
	TON12: TON;
	TON13: TON;
	TON14: TON;
	TON15: TON;
	TON16: TON;
	TON17: TON;
	TON18: TON;
	TON19: TON;
	TON20: TON;
	TON21: TON;
	TON22: TON;
	TON23: TON;
	TON24: TON;
	TON25: TON;
	TON26: TON;
	TON27: TON;
	TON28: TON;
	TON29: TON;
	TON30: TON;
	
END_VAR

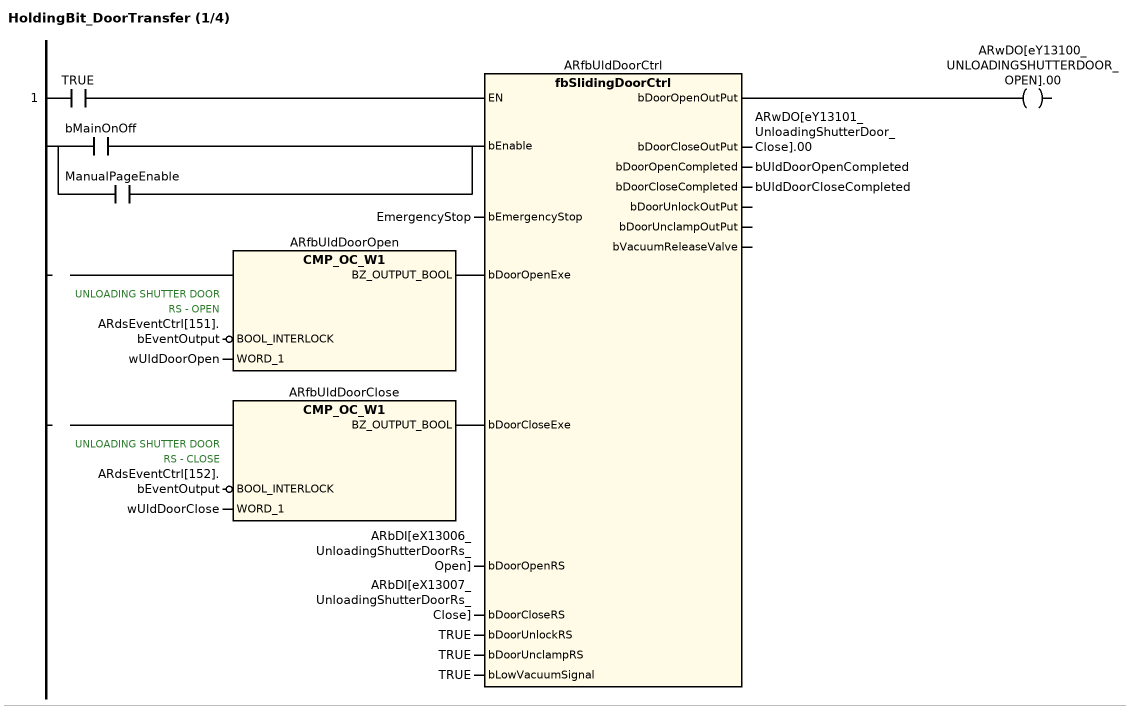
// NETWORK 1
//   ARdsEventCtrl[151].bEventOutput: UNLOADING SHUTTER DOOR RS - OPEN
//   ARdsEventCtrl[152].bEventOutput: UNLOADING SHUTTER DOOR RS - CLOSE
ARfbUldDoorOpen(BOOL_INTERLOCK := NOT ARdsEventCtrl[151].bEventOutput, WORD_1 := wUldDoorOpen); // CMP_OC_W1
ARfbUldDoorClose(BOOL_INTERLOCK := NOT ARdsEventCtrl[152].bEventOutput, WORD_1 := wUldDoorClose); // CMP_OC_W1
ARfbUldDoorCtrl(
    bEnable := bMainOnOff OR ManualPageEnable,
    bEmergencyStop := EmergencyStop,
    bDoorOpenExe := ARfbUldDoorOpen.BZ_OUTPUT_BOOL,
    bDoorCloseExe := ARfbUldDoorClose.BZ_OUTPUT_BOOL,
    bDoorOpenRS := ARbDI[eX13006_UnloadingShutterDoorRs_Open],
    bDoorCloseRS := ARbDI[eX13007_UnloadingShutterDoorRs_Close],
    bDoorUnlockRS := TRUE,
    bDoorUnclampRS := TRUE,
    bLowVacuumSignal := TRUE,
    bDoorCloseOutPut => ARwDO[eY13101_UnloadingShutterDoor_Close].00,
    bDoorOpenCompleted => bUldDoorOpenCompleted,
    bDoorCloseCompleted => bUldDoorCloseCompleted); // fbSlidingDoorCtrl
ARwDO[eY13100_UNLOADINGSHUTTERDOOR_OPEN].00 := ARfbUldDoorCtrl.bDoorOpenOutPut;

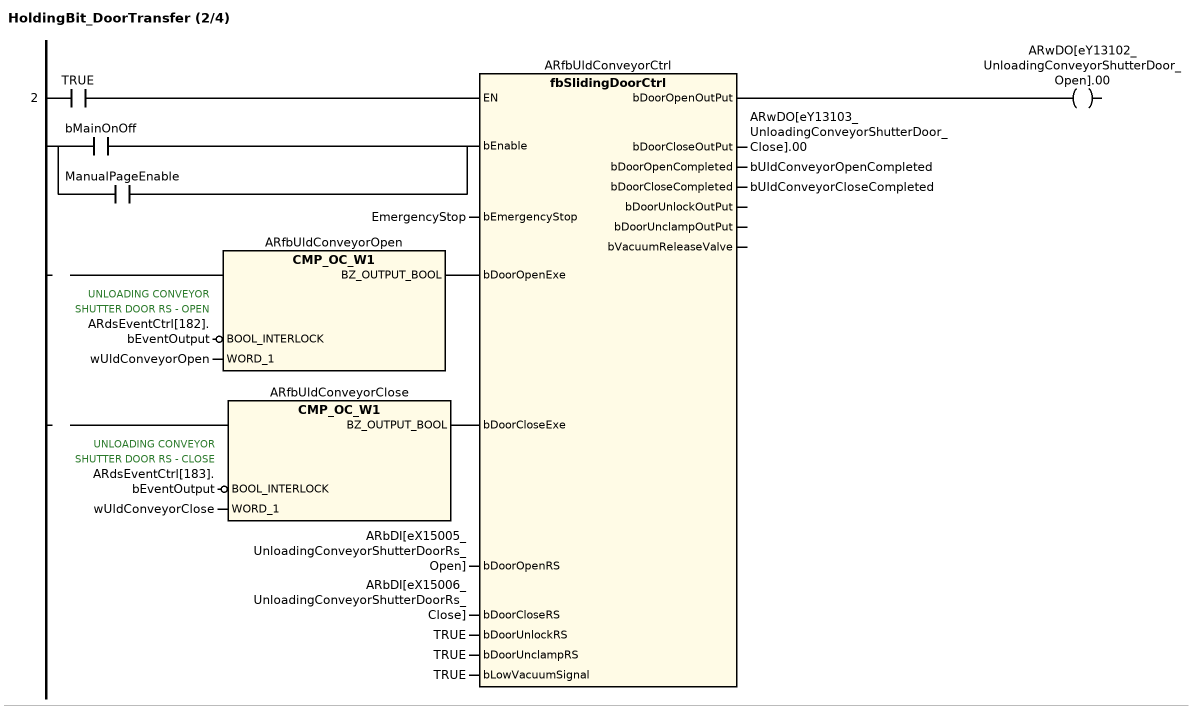
// NETWORK 2
//   ARdsEventCtrl[182].bEventOutput: UNLOADING CONVEYOR SHUTTER DOOR RS - OPEN
//   ARdsEventCtrl[183].bEventOutput: UNLOADING CONVEYOR SHUTTER DOOR RS - CLOSE
ARfbUldConveyorOpen(BOOL_INTERLOCK := NOT ARdsEventCtrl[182].bEventOutput, WORD_1 := wUldConveyorOpen); // CMP_OC_W1
ARfbUldConveyorClose(BOOL_INTERLOCK := NOT ARdsEventCtrl[183].bEventOutput, WORD_1 := wUldConveyorClose); // CMP_OC_W1
ARfbUldConveyorCtrl(
    bEnable := bMainOnOff OR ManualPageEnable,
    bEmergencyStop := EmergencyStop,
    bDoorOpenExe := ARfbUldConveyorOpen.BZ_OUTPUT_BOOL,
    bDoorCloseExe := ARfbUldConveyorClose.BZ_OUTPUT_BOOL,
    bDoorOpenRS := ARbDI[eX15005_UnloadingConveyorShutterDoorRs_Open],
    bDoorCloseRS := ARbDI[eX15006_UnloadingConveyorShutterDoorRs_Close],
    bDoorUnlockRS := TRUE,
    bDoorUnclampRS := TRUE,
    bLowVacuumSignal := TRUE,
    bDoorCloseOutPut => ARwDO[eY13103_UnloadingConveyorShutterDoor_Close].00,
    bDoorOpenCompleted => bUldConveyorOpenCompleted,
    bDoorCloseCompleted => bUldConveyorCloseCompleted); // fbSlidingDoorCtrl
ARwDO[eY13102_UnloadingConveyorShutterDoor_Open].00 := ARfbUldConveyorCtrl.bDoorOpenOutPut;

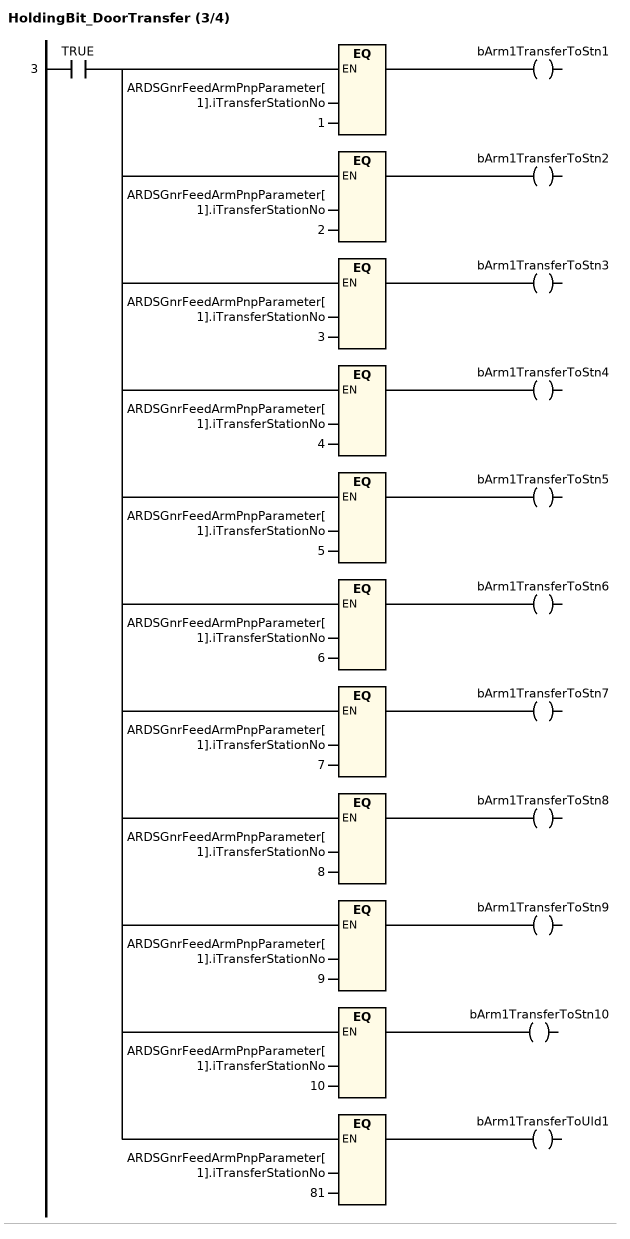
// NETWORK 3
bArm1TransferToStn1 := ARDSGnrFeedArmPnpParameter[1].iTransferStationNo = 1;
bArm1TransferToStn2 := ARDSGnrFeedArmPnpParameter[1].iTransferStationNo = 2;
bArm1TransferToStn3 := ARDSGnrFeedArmPnpParameter[1].iTransferStationNo = 3;
bArm1TransferToStn4 := ARDSGnrFeedArmPnpParameter[1].iTransferStationNo = 4;
bArm1TransferToStn5 := ARDSGnrFeedArmPnpParameter[1].iTransferStationNo = 5;
bArm1TransferToStn6 := ARDSGnrFeedArmPnpParameter[1].iTransferStationNo = 6;
bArm1TransferToStn7 := ARDSGnrFeedArmPnpParameter[1].iTransferStationNo = 7;
bArm1TransferToStn8 := ARDSGnrFeedArmPnpParameter[1].iTransferStationNo = 8;
bArm1TransferToStn9 := ARDSGnrFeedArmPnpParameter[1].iTransferStationNo = 9;
bArm1TransferToStn10 := ARDSGnrFeedArmPnpParameter[1].iTransferStationNo = 10;
bArm1TransferToUld1 := ARDSGnrFeedArmPnpParameter[1].iTransferStationNo = 81;

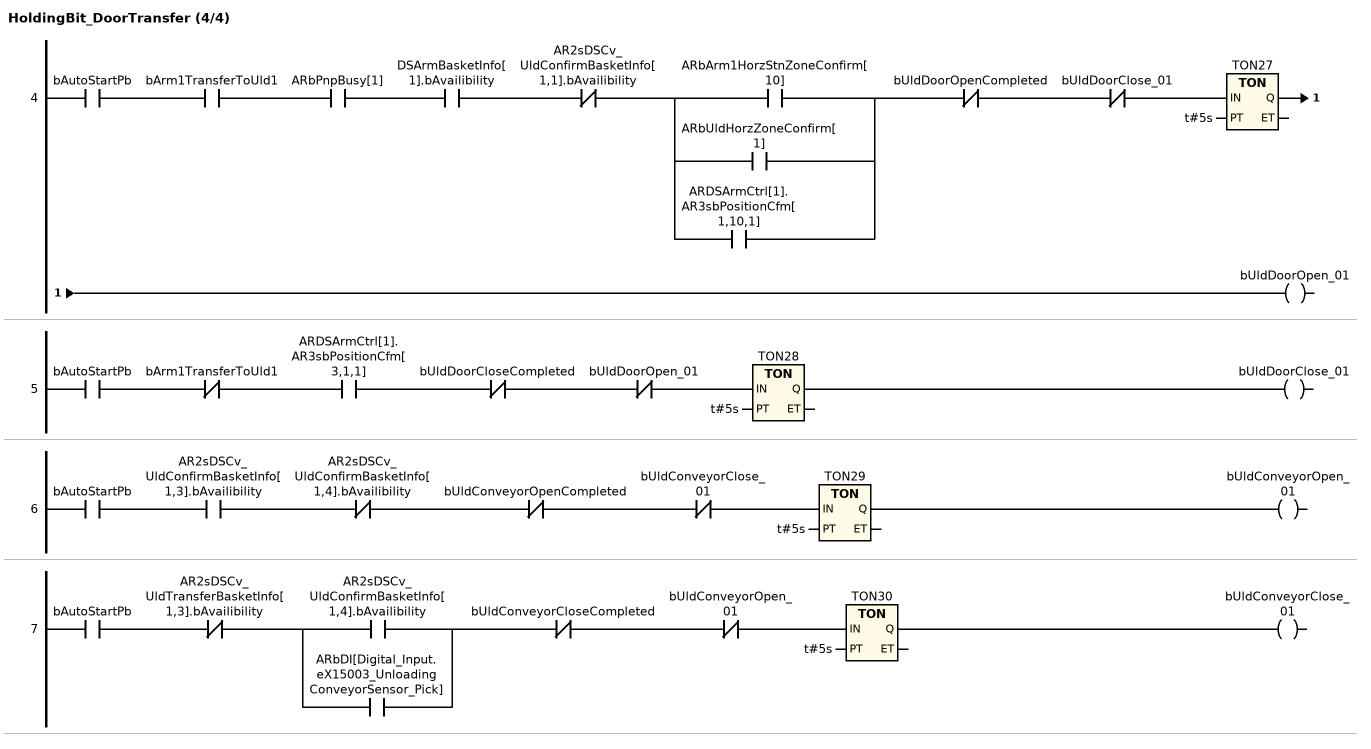
// NETWORK 4
TON27(IN := bAutoStartPb AND bArm1TransferToUld1 AND ARbPnpBusy[1] AND DSArmBasketInfo[1].bAvailibility AND NOT AR2sDSCv_UldConfirmBasketInfo[1,1].bAvailibility AND (ARbArm1HorzStnZoneConfirm[10] OR ARbUldHorzZoneConfirm[1] OR ARDSArmCtrl[1].AR3sbPositionCfm[1,10,1]) AND NOT bUldDoorOpenCompleted AND NOT bUldDoorClose_01, PT := t#5s); // TON
bUldDoorOpen_01 := TON27.Q;

// NETWORK 5
TON28(IN := bAutoStartPb AND NOT bArm1TransferToUld1 AND ARDSArmCtrl[1].AR3sbPositionCfm[3,1,1] AND NOT bUldDoorCloseCompleted AND NOT bUldDoorOpen_01, PT := t#5s); // TON
bUldDoorClose_01 := TON28.Q;

// NETWORK 6
TON29(IN := bAutoStartPb AND AR2sDSCv_UldConfirmBasketInfo[1,3].bAvailibility AND NOT AR2sDSCv_UldConfirmBasketInfo[1,4].bAvailibility AND NOT bUldConveyorOpenCompleted AND NOT bUldConveyorClose_01, PT := t#5s); // TON
bUldConveyorOpen_01 := TON29.Q;

// NETWORK 7
TON30(IN := bAutoStartPb AND NOT AR2sDSCv_UldTransferBasketInfo[1,3].bAvailibility AND (AR2sDSCv_UldConfirmBasketInfo[1,4].bAvailibility OR ARbDI[Digital_Input.eX15003_UnloadingConveyorSensor_Pick]) AND NOT bUldConveyorCloseCompleted AND NOT bUldConveyorOpen_01, PT := t#5s); // TON
bUldConveyorClose_01 := TON30.Q;

END_PROGRAM

// ---- FBs/B_JKS_CustomFB/fbGeneralfbFolder/fbSlidingDoorCtrl.TcPOU
FUNCTION_BLOCK fbSlidingDoorCtrl
VAR_INPUT

	bEnable				: BOOL;
	bEmergencyStop		: BOOL;
	bDoorOpenExe		: BOOL;
	bDoorCloseExe		: BOOL;
	bDoorOpenRS		: BOOL;
	bDoorCloseRS		: BOOL;
	bDoorUnlockRS		: BOOL;
	bDoorUnclampRS		: BOOL;
	bLowVacuumSignal	: BOOL;

END_VAR
VAR_OUTPUT

	bDoorOpenOutPut			: BOOL;
	bDoorCloseOutPut		: BOOL;
	bDoorOpenCompleted		: BOOL;
	bDoorCloseCompleted		: BOOL;
	bDoorUnlockOutPut		: BOOL;
	bDoorUnclampOutPut		: BOOL;
	bVacuumReleaseValve	: BOOL;

END_VAR



VAR
	step1:BOOL;
	step2:BOOL;
	step3:BOOL;
	step4:BOOL;
	step5:BOOL;
	step6:BOOL;


END_VAR

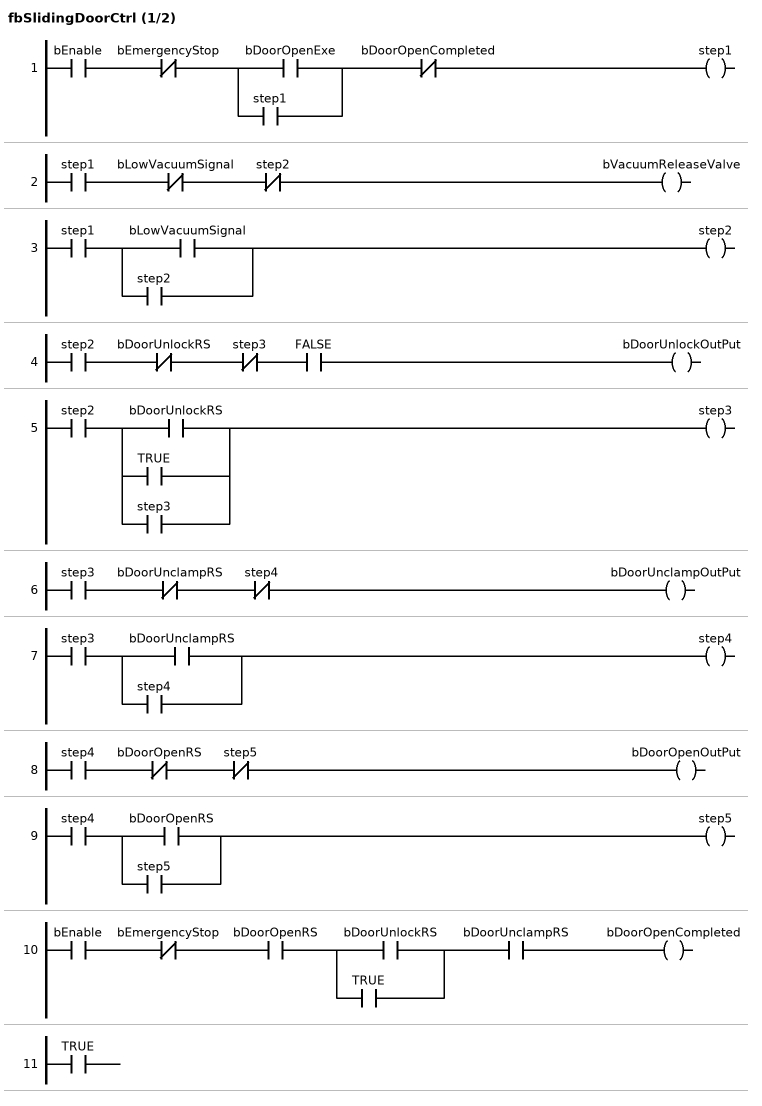
// NETWORK 1
step1 := (bEnable AND NOT bEmergencyStop AND (bDoorOpenExe OR step1)) AND NOT bDoorOpenCompleted;

// NETWORK 2
bVacuumReleaseValve := step1 AND NOT bLowVacuumSignal AND NOT step2;

// NETWORK 3
step2 := step1 AND (bLowVacuumSignal OR step2);

// NETWORK 4
bDoorUnlockOutPut := step2 AND NOT bDoorUnlockRS AND NOT step3 AND FALSE;

// NETWORK 5
step3 := step2 AND (bDoorUnlockRS OR TRUE OR step3);

// NETWORK 6
bDoorUnclampOutPut := step3 AND NOT bDoorUnclampRS AND NOT step4;

// NETWORK 7
step4 := step3 AND (bDoorUnclampRS OR step4);

// NETWORK 8
bDoorOpenOutPut := step4 AND NOT bDoorOpenRS AND NOT step5;

// NETWORK 9
step5 := step4 AND (bDoorOpenRS OR step5);

// NETWORK 10
bDoorOpenCompleted := (bEnable AND NOT bEmergencyStop AND bDoorOpenRS AND (bDoorUnlockRS OR TRUE)) AND bDoorUnclampRS;

// NETWORK 11

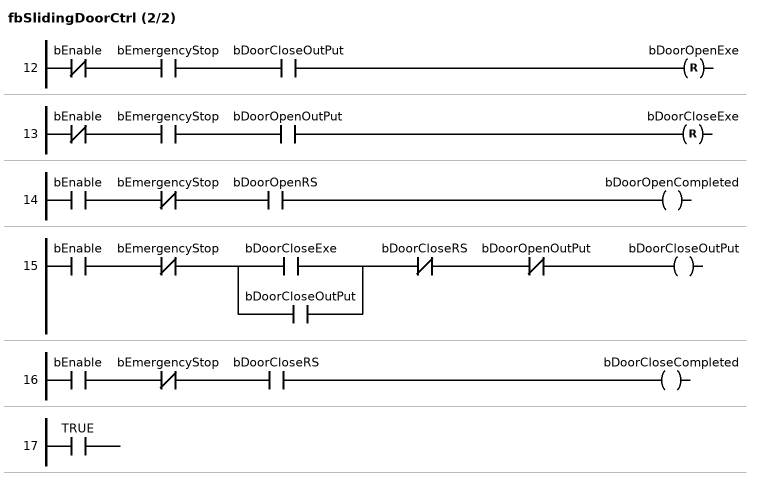
// NETWORK 12
bDoorOpenExe R= NOT bEnable AND bEmergencyStop AND bDoorCloseOutPut;

// NETWORK 13
bDoorCloseExe R= NOT bEnable AND bEmergencyStop AND bDoorOpenOutPut;

// NETWORK 14
bDoorOpenCompleted := bEnable AND NOT bEmergencyStop AND bDoorOpenRS;

// NETWORK 15
bDoorCloseOutPut := (bEnable AND NOT bEmergencyStop AND (bDoorCloseExe OR bDoorCloseOutPut)) AND NOT bDoorCloseRS AND NOT bDoorOpenOutPut;

// NETWORK 16
bDoorCloseCompleted := bEnable AND NOT bEmergencyStop AND bDoorCloseRS;

// NETWORK 17

END_FUNCTION_BLOCK

// ---- FBs/B_JKS_OldFB/Word to Bit/CMP_OC_W1.TcPOU
FUNCTION_BLOCK CMP_OC_W1

VAR_INPUT
	BOOL_INTERLOCK : BOOL; (*INTERLOCK*)
	WORD_1: WORD;		(*WORD 1*)
	END_VAR


VAR_OUTPUT
	BZ_OUTPUT_BOOL : BOOL;
END_VAR


VAR
	OUT_1: BOOL;
END_VAR

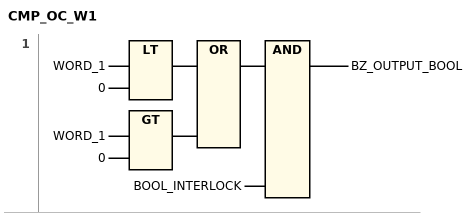
// NETWORK 1
BZ_OUTPUT_BOOL := (WORD_1 < 0 OR WORD_1 > 0) AND BOOL_INTERLOCK;

END_FUNCTION_BLOCK

// ---- POUs/MainProgram/Other/HoldingBitCtrl.TcPOU
PROGRAM HoldingBitCtrl
VAR
	ARfbStnDoorOpenBit : 	ARRAY [1..iStnQty] OF HoldingBitSV;
	ARfbStnDoorCloseBit : 	ARRAY [1..iStnQty] OF HoldingBitSV;

	LdDoorOpenBit: HoldingBitSV;
	LdDoorCloseBit: HoldingBitSV;

	UldDoorOpenBit: HoldingBitSV;
	UldDoorCloseBit: HoldingBitSV;

	ARfbStnDoorClampBit 			: ARRAY [1..iStnQty] OF HoldingBitSV;
	ARfbStnDoorUnclampBit 		: ARRAY [1..iStnQty] OF HoldingBitSV;

	ARfbStnCylinderFrontBit		: ARRAY [1..iStnQty] OF HoldingBitSV;
	ARfbStnCylinderBackBit		: ARRAY [1..iStnQty] OF HoldingBitSV;

	LdConveyorIn : HoldingBitSV;
	LdConveyorOut: HoldingBitSV;

	UldConveyorOpen: HoldingBitSV;
	UldConveyorClose: HoldingBitSV;

	LdConveyorUp: HoldingBitSV;
	LdConveyorDown: HoldingBitSV;

	UldConveyorUp: HoldingBitSV;
	UldConveyorDown: HoldingBitSV;

	NIL: BOOL;

END_VAR

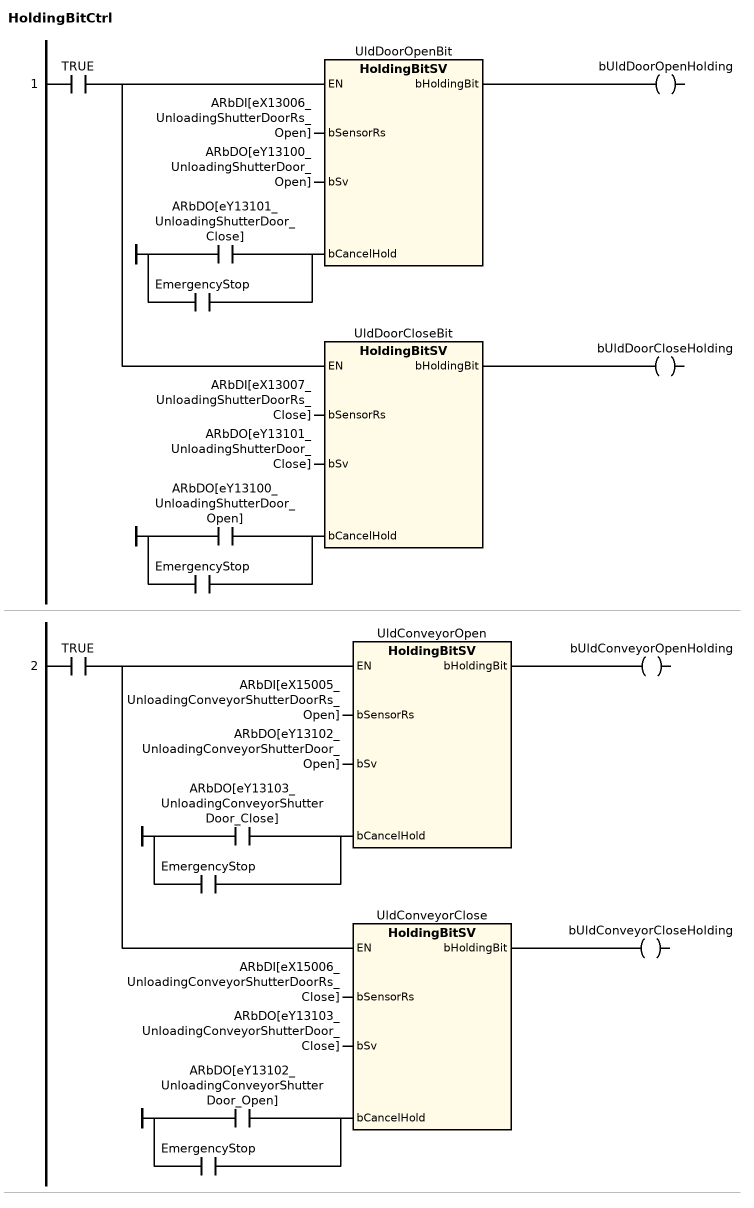
// NETWORK 1
UldDoorOpenBit(
    bSensorRs := ARbDI[eX13006_UnloadingShutterDoorRs_Open],
    bSv := ARbDO[eY13100_UnloadingShutterDoor_Open],
    bCancelHold := ARbDO[eY13101_UnloadingShutterDoor_Close] OR EmergencyStop); // HoldingBitSV
bUldDoorOpenHolding := UldDoorOpenBit.bHoldingBit;
UldDoorCloseBit(
    bSensorRs := ARbDI[eX13007_UnloadingShutterDoorRs_Close],
    bSv := ARbDO[eY13101_UnloadingShutterDoor_Close],
    bCancelHold := ARbDO[eY13100_UnloadingShutterDoor_Open] OR EmergencyStop); // HoldingBitSV
bUldDoorCloseHolding := UldDoorCloseBit.bHoldingBit;

// NETWORK 2
UldConveyorOpen(
    bSensorRs := ARbDI[eX15005_UnloadingConveyorShutterDoorRs_Open],
    bSv := ARbDO[eY13102_UnloadingConveyorShutterDoor_Open],
    bCancelHold := ARbDO[eY13103_UnloadingConveyorShutterDoor_Close] OR EmergencyStop); // HoldingBitSV
bUldConveyorOpenHolding := UldConveyorOpen.bHoldingBit;
UldConveyorClose(
    bSensorRs := ARbDI[eX15006_UnloadingConveyorShutterDoorRs_Close],
    bSv := ARbDO[eY13103_UnloadingConveyorShutterDoor_Close],
    bCancelHold := ARbDO[eY13102_UnloadingConveyorShutterDoor_Open] OR EmergencyStop); // HoldingBitSV
bUldConveyorCloseHolding := UldConveyorClose.bHoldingBit;

END_PROGRAM

// ---- FBs/B_JKS_CustomFB/Other/HoldingBitSV.TcPOU
FUNCTION_BLOCK HoldingBitSV
VAR_INPUT

	bSensorRs:BOOL;
	bSv:BOOL;
	bCancelHold:BOOL;

END_VAR
VAR_OUTPUT

	bHoldingBit:BOOL;

END_VAR
VAR
	SensorComfirm: R_TRIG;
END_VAR

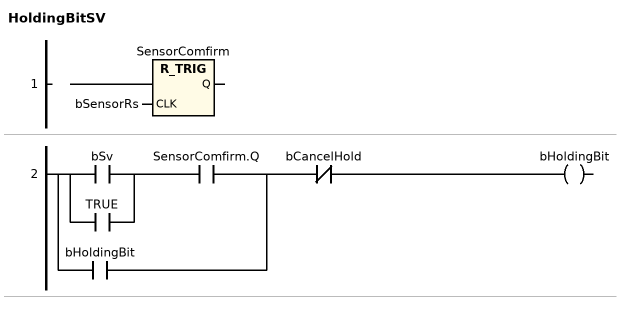
// NETWORK 1
SensorComfirm(CLK := bSensorRs); // R_TRIG

// NETWORK 2
bHoldingBit := ((bSv OR TRUE) AND SensorComfirm.Q OR bHoldingBit) AND NOT bCancelHold;

END_FUNCTION_BLOCK

// ---- POUs/MainProgram/Other/ProHMIMapping.TcPOU
PROGRAM ProHMIMapping
VAR PERSISTENT
	iProductRecipeNo: INT;
	bProductRecipeCopyPB: BOOL;
	iCopyToProductRecipeNo: INT;
	iBufferProductRecipeNo: INT;
	bReadParameter: BOOL;
	DsA1HMInPnpSequenceMemory: DSA1_PnpSequenceMemory;
	bReadDelay: BOOL;
	tReadDelayTimer: TON;
	bTest: BOOL;


	UDSHmiMappingBasketInfo: BOOL;
	HmiMappingBasketInfo: BOOL;

	bWriteParameter: BOOL;
	bWriteDelay: BOOL;
	tWriteDelayTimer: TON;

	iProductRecipeBuffer10: BOOL;

	bWrite2Parameter: BOOL;
	bWrite2Delay: BOOL;
	tWrite2DelayTimer: TON;
	ARiBasketInfo1Buffer: ARRAY [1..30] OF INT;
	ARiBasketInfo2Buffer: ARRAY [1..30] OF INT;
	i16SubTankPumpLPM: BOOL;

(*New*)
	ARiHMIPickStationNo : ARRAY [0..iProductRecipeStepArrayQty] OF INT; (* Byte "n+162~n+223" *)

	ARiHMICallArmNo : ARRAY [0..iProductRecipeStepArrayQty] OF INT; (* Byte "n+100~n+161" *)
	ARiHMITransferStationNo : ARRAY [0..iProductRecipeStepArrayQty] OF INT; (* Byte "n+224~n+285" *)

	ARiHMIStnSeqRepNo : ARRAY [0..iProductRecipeStepArrayQty] OF INT; (* Byte "n+596~n+657" *)

(*Will fix the Value*)
	ARiHMIDownPickPatternNo : ARRAY [0..iProductRecipeStepArrayQty] OF INT; (* Byte "n+286~n+347" *)
	ARiHMIUpPickPatternNo : ARRAY [0..iProductRecipeStepArrayQty] OF INT; (* Byte "n+348~n+409" *)
	ARiHMIDownTransferPatternNo : ARRAY [0..iProductRecipeStepArrayQty] OF INT; (* Byte "n+410~n+471" *)
	ARiHMIUpTransferPatternNo : ARRAY [0..iProductRecipeStepArrayQty] OF INT; (* Byte "n+472~n+533" *)
	ARiHMIRepeatUpDownCycle : ARRAY [0..iProductRecipeStepArrayQty] OF INT; (* Byte "n+534~n+595" *)




	iFixValueFL: INT;
END_VAR
VAR





	iFixValueStepFL: INT;
	iVisibleBitFL: INT;
	iStnProcessStatusFL: INT;

	fbV2HMIStnMinMaxEffTimeDisplay: fbV2_HMIStnMinMaxEffTimeDisplay;


END_VAR

fbV2HMIStnMinMaxEffTimeDisplay(DSStnBasketInfo:= DSStnBasketInfo , ARDsStnMinMaxEffTimeDisplay=> ARDsStnMinMaxEffTimeDisplay );

ARDsStnMinMaxEffTimeDisplay[1].iMinTime;
ARDsStnMinMaxEffTimeDisplay[1].iMaxTime;
ARDsStnMinMaxEffTimeDisplay[1].iEffTime;

ARDsStnMinMaxEffTimeDisplay[2].iMinTime;
ARDsStnMinMaxEffTimeDisplay[2].iMaxTime;
ARDsStnMinMaxEffTimeDisplay[2].iEffTime;

ARDsStnMinMaxEffTimeDisplay[3].iMinTime;
ARDsStnMinMaxEffTimeDisplay[3].iMaxTime;
ARDsStnMinMaxEffTimeDisplay[3].iEffTime;

ARDsStnMinMaxEffTimeDisplay[4].iMinTime;
ARDsStnMinMaxEffTimeDisplay[4].iMaxTime;
ARDsStnMinMaxEffTimeDisplay[4].iEffTime;

ARDsStnMinMaxEffTimeDisplay[5].iMinTime;
ARDsStnMinMaxEffTimeDisplay[5].iMaxTime;
ARDsStnMinMaxEffTimeDisplay[5].iEffTime;

ARDsStnMinMaxEffTimeDisplay[6].iMinTime;
ARDsStnMinMaxEffTimeDisplay[6].iMaxTime;
ARDsStnMinMaxEffTimeDisplay[6].iEffTime;

ARDsStnMinMaxEffTimeDisplay[7].iMinTime;
ARDsStnMinMaxEffTimeDisplay[7].iMaxTime;
ARDsStnMinMaxEffTimeDisplay[7].iEffTime;

ARDsStnMinMaxEffTimeDisplay[8].iMinTime;
ARDsStnMinMaxEffTimeDisplay[8].iMaxTime;
ARDsStnMinMaxEffTimeDisplay[8].iEffTime;

ARDsStnMinMaxEffTimeDisplay[9].iMinTime;
ARDsStnMinMaxEffTimeDisplay[9].iMaxTime;
ARDsStnMinMaxEffTimeDisplay[9].iEffTime;

ARDsStnMinMaxEffTimeDisplay[10].iMinTime;
ARDsStnMinMaxEffTimeDisplay[10].iMaxTime;
ARDsStnMinMaxEffTimeDisplay[10].iEffTime;

ARDsStnMinMaxEffTimeDisplay[11].iMinTime;
ARDsStnMinMaxEffTimeDisplay[11].iMaxTime;
ARDsStnMinMaxEffTimeDisplay[11].iEffTime;

ARDsStnMinMaxEffTimeDisplay[12].iMinTime;
ARDsStnMinMaxEffTimeDisplay[12].iMaxTime;
ARDsStnMinMaxEffTimeDisplay[12].iEffTime;


bRecipeSavePb;

(*
DSA1fbPnpSequenceMemoryStore.iCopyToProductRecipeNo := iCopyToProductRecipeNo;
DSA1fbPnpSequenceMemoryStore.bCopyPB := bProductRecipeCopyPB;
DSA1fbPnpSequenceMemoryStore.iProductRecipeNo := iProductRecipeNo;
*)
IF iProductRecipeNo <> iBufferProductRecipeNo THEN
bReadDelay := TRUE;
END_IF

tReadDelayTimer(IN:=bReadDelay , PT:=t#0.2s , Q=> , ET=> );

IF bReadDelay AND tReadDelayTimer.Q THEN
bReadParameter := TRUE;
iBufferProductRecipeNo := iProductRecipeNo;
bReadDelay := FALSE;
END_IF

IF NOT bReadParameter AND NOT bReadDelay THEN
(*
ARiHMIPickStationNo 			:= DSA1fbPnpSequenceMemoryStore.DsA1inPnpSequenceMemory.ARiPickStationNo;
*)

DSA1fbPnpSequenceMemoryStore.DsA1inPnpSequenceMemory.ARiCallArmNo 				:= ARiHMICallArmNo;                               (*OFF SIGNAL WHEN HAVE TWO ARMs INVOLVED*)

(*DSA1fbPnpSequenceMemoryStore.DsA1inPnpSequenceMemory.ARiTransferStationNo 			:= ARiHMITransferStationNo;
*)
DSA1fbPnpSequenceMemoryStore.DsA1inPnpSequenceMemory.ARiDownPickPatternNo 		:= ARiHMIDownPickPatternNo;
(*DSA1fbPnpSequenceMemoryStore.DsA1inPnpSequenceMemory.ARiUpPickPatternNo 			:= ARiHMIUpPickPatternNo;
DSA1fbPnpSequenceMemoryStore.DsA1inPnpSequenceMemory.ARiDownTransferPatternNo 	:= ARiHMIDownTransferPatternNo;
*)DSA1fbPnpSequenceMemoryStore.DsA1inPnpSequenceMemory.ARiUpTransferPatternNo 		:= ARiHMIUpTransferPatternNo;
DSA1fbPnpSequenceMemoryStore.DsA1inPnpSequenceMemory.ARiRepeatUpDownCycle 		:= ARiHMIRepeatUpDownCycle;
(*DSA1fbPnpSequenceMemoryStore.DsA1inPnpSequenceMemory.ARiStnSeqRepNo 			:= ARiHMIStnSeqRepNo;

DSA1fbPnpSequenceMemoryStore.DsA1inPnpSequenceMemory.sDescription 					:= sProductRecipeDescription;*)
END_IF

IF bReadParameter THEN

(*
ARiHMIPickStationNo 			:= DSA1fbPnpSequenceMemoryStore.DsA1inPnpSequenceMemory.ARiPickStationNo;
*)
ARiHMICallArmNo				:= DSA1fbPnpSequenceMemoryStore.DsA1inPnpSequenceMemory.ARiCallArmNo;                       (*OFF SIGNAL WHEN HAVE TWO ARMs INVOLVED*)
(*ARiHMITransferStationNo		:= DSA1fbPnpSequenceMemoryStore.DsA1inPnpSequenceMemory.ARiTransferStationNo;
*)
ARiHMIDownPickPatternNo		:= DSA1fbPnpSequenceMemoryStore.DsA1inPnpSequenceMemory.ARiDownPickPatternNo;
(*ARiHMIUpPickPatternNo		:= DSA1fbPnpSequenceMemoryStore.DsA1inPnpSequenceMemory.ARiUpPickPatternNo;
ARiHMIDownTransferPatternNo	:= DSA1fbPnpSequenceMemoryStore.DsA1inPnpSequenceMemory.ARiDownTransferPatternNo;
*)ARiHMIUpTransferPatternNo	:= DSA1fbPnpSequenceMemoryStore.DsA1inPnpSequenceMemory.ARiUpTransferPatternNo;
ARiHMIRepeatUpDownCycle	:= DSA1fbPnpSequenceMemoryStore.DsA1inPnpSequenceMemory.ARiRepeatUpDownCycle;
(*ARiHMIStnSeqRepNo			:= DSA1fbPnpSequenceMemoryStore.DsA1inPnpSequenceMemory.ARiStnSeqRepNo;

sProductRecipeDescription := DSA1fbPnpSequenceMemoryStore.DsA1inPnpSequenceMemory.sDescription;*)
bReadParameter := FALSE;
END_IF


(*Fixed Value - No parameter change required*)
iFixValueFL := 0;

	FOR iFixValueFL := 0 TO iProductRecipeStepArrayQty DO
		IF iFixValueFL >= 0 AND iFixValueFL <= iProductRecipeStepArrayQty THEN
			ARiHMIDownPickPatternNo[iFixValueFL] 		:= 1;
			ARiHMIUpPickPatternNo[iFixValueFL]		:= 1;
			ARiHMIDownTransferPatternNo[iFixValueFL] 	:= 1;
			ARiHMIUpTransferPatternNo[iFixValueFL] 	:= 1;
			ARiHMIRepeatUpDownCycle[iFixValueFL] 	:= 1;
			ARiHMICallArmNo[iFixValueFL] 				:= 1;        (*OFF SIGNAL WHEN HAVE TWO ARMs INVOLVED*)

		END_IF

		IF iFixValueFL >= 1 AND iFixValueFL <= iProductRecipeStepArrayQty THEN
			ARDsStnSeqProcessCtrl[1].Out_ARiCurrentCycle[iFixValueFL] 		:= 1;
			ARDsStnSeqProcessCtrl[2].Out_ARiCurrentCycle[iFixValueFL] 		:= 1;
			ARDsStnSeqProcessCtrl[3].Out_ARiCurrentCycle[iFixValueFL] 		:= 1;
			ARDsStnSeqProcessCtrl[4].Out_ARiCurrentCycle[iFixValueFL] 		:= 1;
			ARDsStnSeqProcessCtrl[5].Out_ARiCurrentCycle[iFixValueFL] 		:= 1;
			ARDsStnSeqProcessCtrl[6].Out_ARiCurrentCycle[iFixValueFL] 		:= 1;
			ARDsStnSeqProcessCtrl[7].Out_ARiCurrentCycle[iFixValueFL] 		:= 1;
			ARDsStnSeqProcessCtrl[8].Out_ARiCurrentCycle[iFixValueFL] 		:= 1;
			ARDsStnSeqProcessCtrl[9].Out_ARiCurrentCycle[iFixValueFL] 		:= 1;
			ARDsStnSeqProcessCtrl[10].Out_ARiCurrentCycle[iFixValueFL] 		:= 1;
		END_IF

	END_FOR



(*Read SeqRecipeDescription for display in Product Recipe Page*)

(*Step1*)
IF DSA1fbPnpSequenceMemoryStore.DsA1inPnpSequenceMemory.ARiTransferStationNo[1] >= 1 AND DSA1fbPnpSequenceMemoryStore.DsA1inPnpSequenceMemory.ARiTransferStationNo[1] <= iStnQty THEN
sProductRecipeStep1SeqRecipeDescription :=
fbMainStationProcess_Stn[(**)DSA1fbPnpSequenceMemoryStore.DsA1inPnpSequenceMemory.ARiTransferStationNo[1](**)]
.StnSeqProcessfb.fbStationSequenceRecipefb.ARsStorageStationSequenceRecipeDescription[(**)DSA1fbPnpSequenceMemoryStore.DsA1inPnpSequenceMemory.ARiStnSeqRepNo[1](**)];
ELSE
sProductRecipeStep1SeqRecipeDescription := '';
END_IF

(*Step2*)
IF DSA1fbPnpSequenceMemoryStore.DsA1inPnpSequenceMemory.ARiTransferStationNo[2] >= 1 AND DSA1fbPnpSequenceMemoryStore.DsA1inPnpSequenceMemory.ARiTransferStationNo[2] <= iStnQty THEN
sProductRecipeStep2SeqRecipeDescription :=
fbMainStationProcess_Stn[(**)DSA1fbPnpSequenceMemoryStore.DsA1inPnpSequenceMemory.ARiTransferStationNo[2](**)]
.StnSeqProcessfb.fbStationSequenceRecipefb.ARsStorageStationSequenceRecipeDescription[(**)DSA1fbPnpSequenceMemoryStore.DsA1inPnpSequenceMemory.ARiStnSeqRepNo[2](**)];
ELSE
sProductRecipeStep2SeqRecipeDescription := '';
END_IF

(*Step3*)
IF DSA1fbPnpSequenceMemoryStore.DsA1inPnpSequenceMemory.ARiTransferStationNo[3] >= 1 AND DSA1fbPnpSequenceMemoryStore.DsA1inPnpSequenceMemory.ARiTransferStationNo[3] <= iStnQty THEN
sProductRecipeStep3SeqRecipeDescription :=
fbMainStationProcess_Stn[(**)DSA1fbPnpSequenceMemoryStore.DsA1inPnpSequenceMemory.ARiTransferStationNo[3](**)]
.StnSeqProcessfb.fbStationSequenceRecipefb.ARsStorageStationSequenceRecipeDescription[(**)DSA1fbPnpSequenceMemoryStore.DsA1inPnpSequenceMemory.ARiStnSeqRepNo[3](**)];
ELSE
sProductRecipeStep3SeqRecipeDescription := '';
END_IF

(*Step4*)
IF DSA1fbPnpSequenceMemoryStore.DsA1inPnpSequenceMemory.ARiTransferStationNo[4] >= 1 AND DSA1fbPnpSequenceMemoryStore.DsA1inPnpSequenceMemory.ARiTransferStationNo[4] <= iStnQty THEN
sProductRecipeStep4SeqRecipeDescription :=
fbMainStationProcess_Stn[(**)DSA1fbPnpSequenceMemoryStore.DsA1inPnpSequenceMemory.ARiTransferStationNo[4](**)]
.StnSeqProcessfb.fbStationSequenceRecipefb.ARsStorageStationSequenceRecipeDescription[(**)DSA1fbPnpSequenceMemoryStore.DsA1inPnpSequenceMemory.ARiStnSeqRepNo[4](**)];
ELSE
sProductRecipeStep4SeqRecipeDescription := '';
END_IF

(*Step5*)
IF DSA1fbPnpSequenceMemoryStore.DsA1inPnpSequenceMemory.ARiTransferStationNo[5] >= 1 AND DSA1fbPnpSequenceMemoryStore.DsA1inPnpSequenceMemory.ARiTransferStationNo[5] <= iStnQty THEN
sProductRecipeStep5SeqRecipeDescription :=
fbMainStationProcess_Stn[(**)DSA1fbPnpSequenceMemoryStore.DsA1inPnpSequenceMemory.ARiTransferStationNo[5](**)]
.StnSeqProcessfb.fbStationSequenceRecipefb.ARsStorageStationSequenceRecipeDescription[(**)DSA1fbPnpSequenceMemoryStore.DsA1inPnpSequenceMemory.ARiStnSeqRepNo[5](**)];
ELSE
sProductRecipeStep5SeqRecipeDescription := '';
END_IF

(*Step6*)
IF DSA1fbPnpSequenceMemoryStore.DsA1inPnpSequenceMemory.ARiTransferStationNo[6] >= 1 AND DSA1fbPnpSequenceMemoryStore.DsA1inPnpSequenceMemory.ARiTransferStationNo[6] <= iStnQty THEN
sProductRecipeStep6SeqRecipeDescription :=
fbMainStationProcess_Stn[(**)DSA1fbPnpSequenceMemoryStore.DsA1inPnpSequenceMemory.ARiTransferStationNo[6](**)]
.StnSeqProcessfb.fbStationSequenceRecipefb.ARsStorageStationSequenceRecipeDescription[(**)DSA1fbPnpSequenceMemoryStore.DsA1inPnpSequenceMemory.ARiStnSeqRepNo[6](**)];
ELSE
sProductRecipeStep6SeqRecipeDescription := '';
END_IF

(*Step7*)
IF DSA1fbPnpSequenceMemoryStore.DsA1inPnpSequenceMemory.ARiTransferStationNo[7] >= 1 AND DSA1fbPnpSequenceMemoryStore.DsA1inPnpSequenceMemory.ARiTransferStationNo[7] <= iStnQty THEN
sProductRecipeStep7SeqRecipeDescription :=
fbMainStationProcess_Stn[(**)DSA1fbPnpSequenceMemoryStore.DsA1inPnpSequenceMemory.ARiTransferStationNo[7](**)]
.StnSeqProcessfb.fbStationSequenceRecipefb.ARsStorageStationSequenceRecipeDescription[(**)DSA1fbPnpSequenceMemoryStore.DsA1inPnpSequenceMemory.ARiStnSeqRepNo[7](**)];
ELSE
sProductRecipeStep7SeqRecipeDescription := '';
END_IF

(*Step8*)
IF DSA1fbPnpSequenceMemoryStore.DsA1inPnpSequenceMemory.ARiTransferStationNo[8] >= 1 AND DSA1fbPnpSequenceMemoryStore.DsA1inPnpSequenceMemory.ARiTransferStationNo[8] <= iStnQty THEN
sProductRecipeStep8SeqRecipeDescription :=
fbMainStationProcess_Stn[(**)DSA1fbPnpSequenceMemoryStore.DsA1inPnpSequenceMemory.ARiTransferStationNo[8](**)]
.StnSeqProcessfb.fbStationSequenceRecipefb.ARsStorageStationSequenceRecipeDescription[(**)DSA1fbPnpSequenceMemoryStore.DsA1inPnpSequenceMemory.ARiStnSeqRepNo[8](**)];
ELSE
sProductRecipeStep8SeqRecipeDescription := '';
END_IF

(*Step9*)
IF DSA1fbPnpSequenceMemoryStore.DsA1inPnpSequenceMemory.ARiTransferStationNo[9] >= 1 AND DSA1fbPnpSequenceMemoryStore.DsA1inPnpSequenceMemory.ARiTransferStationNo[9] <= iStnQty THEN
sProductRecipeStep9SeqRecipeDescription :=
fbMainStationProcess_Stn[(**)DSA1fbPnpSequenceMemoryStore.DsA1inPnpSequenceMemory.ARiTransferStationNo[9](**)]
.StnSeqProcessfb.fbStationSequenceRecipefb.ARsStorageStationSequenceRecipeDescription[(**)DSA1fbPnpSequenceMemoryStore.DsA1inPnpSequenceMemory.ARiStnSeqRepNo[9](**)];
ELSE
sProductRecipeStep9SeqRecipeDescription := '';
END_IF

(*Step10*)
IF DSA1fbPnpSequenceMemoryStore.DsA1inPnpSequenceMemory.ARiTransferStationNo[10] >= 1 AND DSA1fbPnpSequenceMemoryStore.DsA1inPnpSequenceMemory.ARiTransferStationNo[10] <= iStnQty THEN
sProductRecipeStep10SeqRecipeDescription :=
fbMainStationProcess_Stn[(**)DSA1fbPnpSequenceMemoryStore.DsA1inPnpSequenceMemory.ARiTransferStationNo[10](**)]
.StnSeqProcessfb.fbStationSequenceRecipefb.ARsStorageStationSequenceRecipeDescription[(**)DSA1fbPnpSequenceMemoryStore.DsA1inPnpSequenceMemory.ARiStnSeqRepNo[10](**)];
ELSE
sProductRecipeStep10SeqRecipeDescription := '';
END_IF

(*Step11*)
IF DSA1fbPnpSequenceMemoryStore.DsA1inPnpSequenceMemory.ARiTransferStationNo[11] >= 1 AND DSA1fbPnpSequenceMemoryStore.DsA1inPnpSequenceMemory.ARiTransferStationNo[11] <= iStnQty THEN
sProductRecipeStep11SeqRecipeDescription :=
fbMainStationProcess_Stn[(**)DSA1fbPnpSequenceMemoryStore.DsA1inPnpSequenceMemory.ARiTransferStationNo[11](**)]
.StnSeqProcessfb.fbStationSequenceRecipefb.ARsStorageStationSequenceRecipeDescription[(**)DSA1fbPnpSequenceMemoryStore.DsA1inPnpSequenceMemory.ARiStnSeqRepNo[11](**)];
ELSE
sProductRecipeStep11SeqRecipeDescription := '';
END_IF

(*Step12*)
IF DSA1fbPnpSequenceMemoryStore.DsA1inPnpSequenceMemory.ARiTransferStationNo[12] >= 1 AND DSA1fbPnpSequenceMemoryStore.DsA1inPnpSequenceMemory.ARiTransferStationNo[12] <= iStnQty THEN
sProductRecipeStep12SeqRecipeDescription :=
fbMainStationProcess_Stn[(**)DSA1fbPnpSequenceMemoryStore.DsA1inPnpSequenceMemory.ARiTransferStationNo[12](**)]
.StnSeqProcessfb.fbStationSequenceRecipefb.ARsStorageStationSequenceRecipeDescription[(**)DSA1fbPnpSequenceMemoryStore.DsA1inPnpSequenceMemory.ARiStnSeqRepNo[12](**)];
ELSE
sProductRecipeStep12SeqRecipeDescription := '';
END_IF

(*Step13*)
IF DSA1fbPnpSequenceMemoryStore.DsA1inPnpSequenceMemory.ARiTransferStationNo[13] >= 1 AND DSA1fbPnpSequenceMemoryStore.DsA1inPnpSequenceMemory.ARiTransferStationNo[13] <= iStnQty THEN
sProductRecipeStep13SeqRecipeDescription :=
fbMainStationProcess_Stn[(**)DSA1fbPnpSequenceMemoryStore.DsA1inPnpSequenceMemory.ARiTransferStationNo[13](**)]
.StnSeqProcessfb.fbStationSequenceRecipefb.ARsStorageStationSequenceRecipeDescription[(**)DSA1fbPnpSequenceMemoryStore.DsA1inPnpSequenceMemory.ARiStnSeqRepNo[13](**)];
ELSE
sProductRecipeStep13SeqRecipeDescription := '';
END_IF

(*Step14*)
IF DSA1fbPnpSequenceMemoryStore.DsA1inPnpSequenceMemory.ARiTransferStationNo[14] >= 1 AND DSA1fbPnpSequenceMemoryStore.DsA1inPnpSequenceMemory.ARiTransferStationNo[14] <= iStnQty THEN
sProductRecipeStep14SeqRecipeDescription :=
fbMainStationProcess_Stn[(**)DSA1fbPnpSequenceMemoryStore.DsA1inPnpSequenceMemory.ARiTransferStationNo[14](**)]
.StnSeqProcessfb.fbStationSequenceRecipefb.ARsStorageStationSequenceRecipeDescription[(**)DSA1fbPnpSequenceMemoryStore.DsA1inPnpSequenceMemory.ARiStnSeqRepNo[14](**)];
ELSE
sProductRecipeStep14SeqRecipeDescription := '';
END_IF

(*Step15*)
IF DSA1fbPnpSequenceMemoryStore.DsA1inPnpSequenceMemory.ARiTransferStationNo[15] >= 1 AND DSA1fbPnpSequenceMemoryStore.DsA1inPnpSequenceMemory.ARiTransferStationNo[15] <= iStnQty THEN
sProductRecipeStep15SeqRecipeDescription :=
fbMainStationProcess_Stn[(**)DSA1fbPnpSequenceMemoryStore.DsA1inPnpSequenceMemory.ARiTransferStationNo[15](**)]
.StnSeqProcessfb.fbStationSequenceRecipefb.ARsStorageStationSequenceRecipeDescription[(**)DSA1fbPnpSequenceMemoryStore.DsA1inPnpSequenceMemory.ARiStnSeqRepNo[15](**)];
ELSE
sProductRecipeStep15SeqRecipeDescription := '';
END_IF


(*Generate Visible Bit for Indusoft*)
iVisibleBitFL := 1;

IF iVisibleBitFL >= 1 AND iVisibleBitFL <= iProductRecipeStepArrayQty THEN
	FOR iVisibleBitFL := 1 TO iProductRecipeStepArrayQty DO

		ARbStnSeqRepNoVisible[iVisibleBitFL] := TRUE;

	END_FOR
END_IF


iVisibleBitFL := 1;


IF iVisibleBitFL >= 1 AND iVisibleBitFL <= iProductRecipeStepArrayQty THEN
	FOR iVisibleBitFL := 2 TO iProductRecipeStepArrayQty DO

		IF (DSA1fbPnpSequenceMemoryStore.DsA1inPnpSequenceMemory.ARiTransferStationNo[iVisibleBitFL-1] = ARiUldStnID[1] (*OR DSA1fbPnpSequenceMemoryStore.DsA1inPnpSequenceMemory.ARiTransferStationNo[iVisibleBitFL-1] = ARiUldStnID[2]*))
		OR NOT ARbStnSeqRepNoVisible[iVisibleBitFL-1] THEN
		ARbStnSeqRepNoVisible[iVisibleBitFL] := FALSE;
		END_IF

	END_FOR
END_IF



(*Generate Station - Process Status String for Indusoft*)

iStnProcessStatusFL := 1;


IF iStnProcessStatusFL >= 1 AND iStnProcessStatusFL <= iStnQty THEN
	FOR iStnProcessStatusFL := 1 TO iStnQty DO

		IF DSHmiStationDisplayInfo[iStnProcessStatusFL].bCallArmSpeedProfileMemoryErr
		THEN ARsStnProcessStatus[iStnProcessStatusFL] := 'Arm Speed Profile Memory Error';

		ELSIF DSHmiStationDisplayInfo[iStnProcessStatusFL].bCallPickStationNoErr
		THEN ARsStnProcessStatus[iStnProcessStatusFL] := 'Call Pick Station No Error';

		ELSIF DSHmiStationDisplayInfo[iStnProcessStatusFL].bCallStnSeqRecipeErr
		THEN ARsStnProcessStatus[iStnProcessStatusFL] := 'Call Station Sequence Recipe Error';

		ELSIF DSHmiStationDisplayInfo[iStnProcessStatusFL].bCallTransferStationNoErr
		THEN ARsStnProcessStatus[iStnProcessStatusFL] := 'Call Transfer Station No Error';

		ELSIF DSHmiStationDisplayInfo[iStnProcessStatusFL].bCallUpDownPatternMemoryErr
		THEN ARsStnProcessStatus[iStnProcessStatusFL] := 'Call Up Down Pattern Memory Error';

		ELSIF DSHmiStationDisplayInfo[iStnProcessStatusFL].bInvalidProcessStepErr
		THEN ARsStnProcessStatus[iStnProcessStatusFL] := 'Step Error - Invalid Process Step';

		ELSIF DSHmiStationDisplayInfo[iStnProcessStatusFL].bInvalidProductRecipeNoErr
		THEN ARsStnProcessStatus[iStnProcessStatusFL] := 'Product Recipe Invalid';

		ELSIF DSHmiStationDisplayInfo[iStnProcessStatusFL].bInvalidProductRecipeStepErr
		THEN ARsStnProcessStatus[iStnProcessStatusFL] := 'Product Recipe Step Error';

		ELSIF DSHmiStationDisplayInfo[iStnProcessStatusFL].bStationSequenceProcessCompleted
		THEN ARsStnProcessStatus[iStnProcessStatusFL] := 'Process Completed';

		ELSIF DSHmiStationDisplayInfo[iStnProcessStatusFL].bStationSequenceProcessInProgressFlag
		THEN ARsStnProcessStatus[iStnProcessStatusFL] := 'Process In Progress';

		ELSIF DSHmiStationDisplayInfo[iStnProcessStatusFL].bStationSequenceProcessStart
		THEN ARsStnProcessStatus[iStnProcessStatusFL] := 'Process Start';

		ELSE
			ARsStnProcessStatus[iStnProcessStatusFL] := 'No Process';
		END_IF


	END_FOR
END_IF

END_PROGRAM

// ---- FBs/B_JKS_NewFB_V2/FBP-MTBSubFB/fbV2_HMIStnMinMaxEffTimeDisplay.TcPOU
FUNCTION_BLOCK fbV2_HMIStnMinMaxEffTimeDisplay
VAR_INPUT
	DSStnBasketInfo						: ARRAY [0..iStnQty] OF DSV2_BasketInfo;

END_VAR
VAR_OUTPUT
	ARDsStnMinMaxEffTimeDisplay			:ARRAY [0..iStnQty] OF DSV2_StnMinMaxEffTIme;
END_VAR
VAR
	iMinMaxFL: INT;
END_VAR

iMinMaxFL := 1;
	IF iMinMaxFL >= 1 AND iMinMaxFL <= iStnQty THEN
		FOR iMinMaxFL := 1 TO iStnQty DO

			IF DSStnBasketInfo[iMinMaxFL].bAvailibility THEN
			ARDsStnMinMaxEffTimeDisplay[iMinMaxFL].iMinTime := DSStnBasketInfo[iMinMaxFL].DSV2MinMaxEffTime.ARiMinTime[DSStnBasketInfo[iMinMaxFL].iProductRecipeStepNo];
			ARDsStnMinMaxEffTimeDisplay[iMinMaxFL].iMaxTime := DSStnBasketInfo[iMinMaxFL].DSV2MinMaxEffTime.ARiMaxTime[DSStnBasketInfo[iMinMaxFL].iProductRecipeStepNo];
			ARDsStnMinMaxEffTimeDisplay[iMinMaxFL].iEffTime := DSStnBasketInfo[iMinMaxFL].DSV2MinMaxEffTime.ARiEffTime[DSStnBasketInfo[iMinMaxFL].iProductRecipeStepNo];
			ELSE
			ARDsStnMinMaxEffTimeDisplay[iMinMaxFL].iMinTime := 0;
			ARDsStnMinMaxEffTimeDisplay[iMinMaxFL].iMaxTime := 0;
			ARDsStnMinMaxEffTimeDisplay[iMinMaxFL].iEffTime := 0;
			END_IF
		END_FOR
	END_IF

END_FUNCTION_BLOCK

// ---- POUs/MainProgram/Other/TactTime.TcPOU
PROGRAM TactTime
VAR

	TactTime: TactTimeFB;

END_VAR

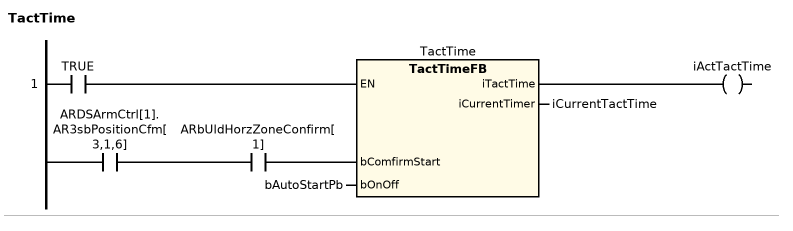
// NETWORK 1
TactTime(
    bComfirmStart := ARDSArmCtrl[1].AR3sbPositionCfm[3,1,6] AND ARbUldHorzZoneConfirm[1],
    bOnOff := bAutoStartPb,
    iCurrentTimer => iCurrentTactTime); // TactTimeFB
iActTactTime := TactTime.iTactTime;

END_PROGRAM

// ---- FBs/B_JKS_CustomFB/Other/TactTimeFB.TcPOU
FUNCTION_BLOCK TactTimeFB
VAR_INPUT
	bComfirmStart:BOOL;
	bOnOff:BOOL;



END_VAR
VAR_OUTPUT
	iTactTime:INT;
	iCurrentTimer:INT;


END_VAR
VAR
	StartCount: BOOL;
	ComfirmPulse: R_TRIG;
	clockPulse: BOOL;
	SecondPulse: CLOCK_PLS;
	AddPulse: R_TRIG;
	currentTimer: INT;
	delayOn: TON;
	PulseOffCount: R_TRIG;
	TimeReset: BOOL;
	DelayTimeron: TON;
	off: BOOL;
	DelayMove: TON;
	movetrig: R_TRIG;
END_VAR
VAR // added by the converter: edge detectors and wires of the graphical bodies
    _w1, _w3 : INT;
    _w2 : ANY;
END_VAR

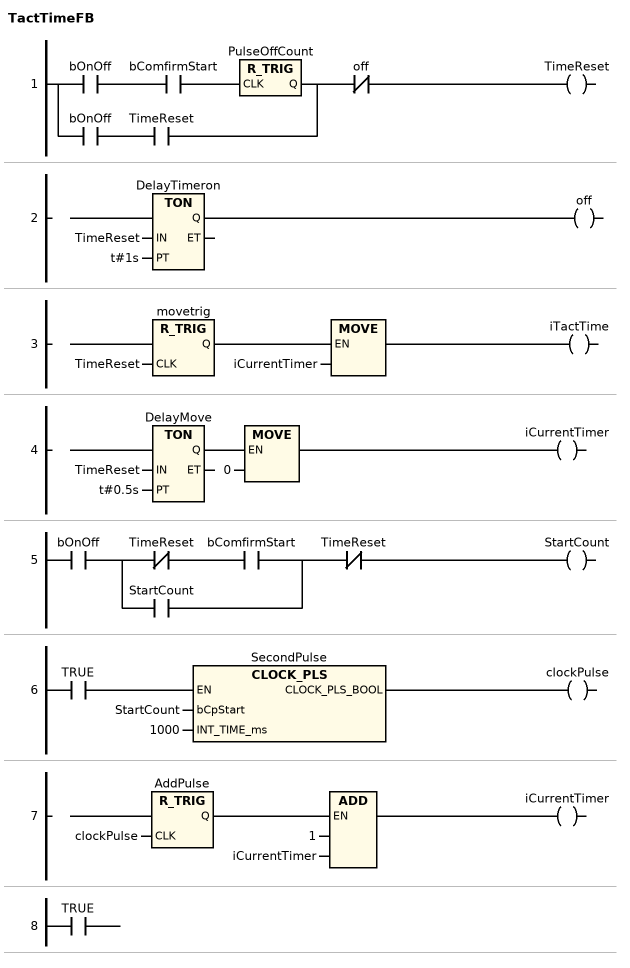
// NETWORK 1
PulseOffCount(CLK := bOnOff AND bComfirmStart); // R_TRIG
TimeReset := (PulseOffCount.Q OR bOnOff AND TimeReset) AND NOT off;

// NETWORK 2
DelayTimeron(IN := TimeReset, PT := t#1s); // TON
off := DelayTimeron.Q;

// NETWORK 3
movetrig(CLK := TimeReset); // R_TRIG
IF movetrig.Q THEN _w1 := iCurrentTimer; END_IF
iTactTime := _w1;

// NETWORK 4
DelayMove(IN := TimeReset, PT := t#0.5s); // TON
IF DelayMove.Q THEN _w2 := 0; END_IF
iCurrentTimer := _w2;

// NETWORK 5
StartCount := (bOnOff AND (NOT TimeReset AND bComfirmStart OR StartCount)) AND NOT TimeReset;

// NETWORK 6
SecondPulse(bCpStart := StartCount, INT_TIME_ms := 1000); // CLOCK_PLS
clockPulse := SecondPulse.CLOCK_PLS_BOOL;

// NETWORK 7
AddPulse(CLK := clockPulse); // R_TRIG
IF AddPulse.Q THEN _w3 := 1 + iCurrentTimer; END_IF
iCurrentTimer := _w3;

// NETWORK 8

END_FUNCTION_BLOCK

// ---- POUs/MainProgram/Other/zHMIMaxMinLimit.TcPOU
PROGRAM zHMIMaxMinLimit
VAR

	iStnFL: INT;
	iArmFL: INT;
	i7DFL: INT;
	iArmSlowPullFL: INT;
	iIRHeaterFL : INT;
END_VAR

(*VacuumPumpLimitAlarmSetMonitoring*) (*For VacPump*)
(*=========================================================*)
(*
iStnFL := 1;
FOR iStnFL := 1 TO iStnQty DO
	IF iStnFL >= 1 AND iStnFL <= iStnQty THEN

		IF  ARdiVacPump1stLimitTimerSV[iStnFL] > 1500 	THEN ARdiVacPump1stLimitTimerSV[iStnFL] := 1500; 	ELSIF ARdiVacPump1stLimitTimerSV[iStnFL] < 1 	THEN ARdiVacPump1stLimitTimerSV[iStnFL] := 1; 	END_IF
		IF  ARdiVacPump2ndLimitTimerSV[iStnFL] > 2000 	THEN ARdiVacPump2ndLimitTimerSV[iStnFL] := 2000; 	ELSIF ARdiVacPump2ndLimitTimerSV[iStnFL] < 1 	THEN ARdiVacPump2ndLimitTimerSV[iStnFL] := 1; 	END_IF

	END_IF
END_FOR
*)

(*StnBasketCounterLimitAlarmSetMonitoring*)
(*=========================================================*)
IF ARdiStnBasketCounter1stLimitSV[1] > 9999 THEN ARdiStnBasketCounter1stLimitSV[1] := 9999; ELSIF ARdiStnBasketCounter1stLimitSV[1] < 1 THEN ARdiStnBasketCounter1stLimitSV[1] := 1; END_IF
IF ARdiStnBasketCounter2ndLimitSV[1] > 9999 THEN ARdiStnBasketCounter2ndLimitSV[1] := 9999; ELSIF ARdiStnBasketCounter2ndLimitSV[1] < 1 THEN ARdiStnBasketCounter2ndLimitSV[1] := 1; END_IF

IF ARdiStnBasketCounter1stLimitSV[2] > 9999 THEN ARdiStnBasketCounter1stLimitSV[2] := 9999; ELSIF ARdiStnBasketCounter1stLimitSV[2] < 1 THEN ARdiStnBasketCounter1stLimitSV[2] := 1; END_IF
IF ARdiStnBasketCounter2ndLimitSV[2] > 9999 THEN ARdiStnBasketCounter2ndLimitSV[2] := 9999; ELSIF ARdiStnBasketCounter2ndLimitSV[2] < 1 THEN ARdiStnBasketCounter2ndLimitSV[2] := 1; END_IF


(*AllStationCallArmTime*)
(*=========================================================*)
IF  tAllStnArmTake > 50 THEN tAllStnArmTake := 50; ELSIF tAllStnArmTake < 10 THEN tAllStnArmTake := 10; END_IF


(*UnloadingBasketConfirmBuzzerTimer*)
(*=========================================================*)
IF  diUnloadingTimer > 999 THEN diUnloadingTimer := 999; ELSIF diUnloadingTimer < 10 THEN diUnloadingTimer := 10; END_IF
IF  diUnloadingSingleBasketReachedTimer > 999 THEN diUnloadingSingleBasketReachedTimer := 999; ELSIF diUnloadingSingleBasketReachedTimer < 10 THEN diUnloadingSingleBasketReachedTimer := 10; END_IF
IF  diUnloadingBuzzerOffHeaterTimer > 999 THEN diUnloadingBuzzerOffHeaterTimer := 999; ELSIF diUnloadingBuzzerOffHeaterTimer < 10 THEN diUnloadingBuzzerOffHeaterTimer := 10; END_IF


(*Flow Box Delay Timer Ctrl*)
(*=========================================================*)
IF  iFFUDelayOffTimerSV_min > 6000 THEN iFFUDelayOffTimerSV_min := 6000; ELSIF iFFUDelayOffTimerSV_min < 60 THEN iFFUDelayOffTimerSV_min := 60; END_IF

(*Agitation Mechanism Delay Timer Ctrl*)
(*=========================================================*)
IF  iStnAgitation1DelayOffTimerSV_min > 60 		THEN iStnAgitation1DelayOffTimerSV_min := 60; 		ELSIF iStnAgitation1DelayOffTimerSV_min < 0 		THEN iStnAgitation1DelayOffTimerSV_min := 0; END_IF
IF  iStnAgitation2DelayOffTimerSV_min > 60 		THEN iStnAgitation2DelayOffTimerSV_min := 60; 		ELSIF iStnAgitation2DelayOffTimerSV_min < 0 		THEN iStnAgitation2DelayOffTimerSV_min := 0; END_IF


(*7 Days AutoMachineOnOff Limit Ctrl*)
(*=========================================================*)
i7DFL := 1;
FOR i7DFL := 1 TO 7 DO
	IF i7DFL >= 1 AND i7DFL <= 7 THEN

		IF  ArwDayOnMinute_IN[i7DFL] > 59 	THEN ArwDayOnMinute_IN[i7DFL] := 59; 	ELSIF ArwDayOnMinute_IN[i7DFL] < 0 	THEN ArwDayOnMinute_IN[i7DFL] := 0; 	END_IF
		IF  ArwDayOffMinute_IN[i7DFL] > 59 	THEN ArwDayOffMinute_IN[i7DFL] := 59; 	ELSIF ArwDayOffMinute_IN[i7DFL] < 0 	THEN ArwDayOffMinute_IN[i7DFL] := 0; 	END_IF
		IF  ArwDayOnHour_IN[i7DFL] > 23 	THEN ArwDayOnHour_IN[i7DFL] := 23; 	ELSIF ArwDayOnHour_IN[i7DFL] < 0 		THEN ArwDayOnHour_IN[i7DFL] := 0; 	END_IF
		IF  ArwDayOffHour_IN[i7DFL] > 23 	THEN ArwDayOffHour_IN[i7DFL] := 23; 	ELSIF ArwDayOffHour_IN[i7DFL] < 0 		THEN ArwDayOffHour_IN[i7DFL] := 0; 	END_IF

	END_IF
END_FOR


(*Conductivity 1st Limit, 2nd Limit Alarm Control*)
(*=========================================================*)
iStnFL := 1;
FOR iStnFL := 1 TO iStnQty DO
	IF iStnFL >= 1 AND iStnFL <= iStnQty THEN

		IF  ARrStnConductivity1stLimitSv[iStnFL] > 9999 THEN ARrStnConductivity1stLimitSv[iStnFL] := 9999; ELSIF ARrStnConductivity1stLimitSv[iStnFL] < 0 THEN ARrStnConductivity1stLimitSv[iStnFL] := 0; END_IF
		IF  ARrStnConductivity2ndLimitSv[iStnFL] > 9999 THEN ARrStnConductivity2ndLimitSv[iStnFL] := 9999; ELSIF ARrStnConductivity2ndLimitSv[iStnFL] < 0 THEN ARrStnConductivity2ndLimitSv[iStnFL] := 0; END_IF
		IF  ARrStnLowConductivitySv[iStnFL] > 99999 THEN ARrStnLowConductivitySv[iStnFL] := 99999; ELSIF ARrStnLowConductivitySv[iStnFL] < 0 THEN ARrStnLowConductivitySv[iStnFL] := 0; END_IF
		IF  ARrStnHighConductivitySv[iStnFL] > 99999 THEN ARrStnHighConductivitySv[iStnFL] := 99999; ELSIF ARrStnHighConductivitySv[iStnFL] < 0 THEN ARrStnHighConductivitySv[iStnFL] := 0; END_IF

	END_IF
END_FOR


(*Ultrasonic Manual Power Setting Control*) (*For Fix Power*)
(*=========================================================*)
iStnFL := 1;
FOR iStnFL := 1 TO iStnQty DO
	IF iStnFL >= 1 AND iStnFL <= iStnQty THEN

		IF  ARiStnManualUSBtmAsv[iStnFL] > 100 THEN ARiStnManualUSBtmAsv[iStnFL] := 100; ELSIF ARiStnManualUSBtmAsv[iStnFL] < 10 THEN ARiStnManualUSBtmAsv[iStnFL] := 10; END_IF
		IF  ARiStnManualUSBtmBsv[iStnFL] > 100 THEN ARiStnManualUSBtmBsv[iStnFL] := 100; ELSIF ARiStnManualUSBtmBsv[iStnFL] < 10 THEN ARiStnManualUSBtmBsv[iStnFL] := 10; END_IF
		IF  ARiStnManualUSBtmCsv[iStnFL] > 100 THEN ARiStnManualUSBtmCsv[iStnFL] := 100; ELSIF ARiStnManualUSBtmCsv[iStnFL] < 10 THEN ARiStnManualUSBtmCsv[iStnFL] := 10; END_IF
		IF  ARiStnManualUSBtmDsv[iStnFL] > 100 THEN ARiStnManualUSBtmDsv[iStnFL] := 100; ELSIF ARiStnManualUSBtmDsv[iStnFL] < 10 THEN ARiStnManualUSBtmDsv[iStnFL] := 10; END_IF

		IF  ARiStnManualUSSideAsv[iStnFL] > 100 THEN ARiStnManualUSSideAsv[iStnFL] := 100; ELSIF ARiStnManualUSSideAsv[iStnFL] < 10 THEN ARiStnManualUSSideAsv[iStnFL] := 10; END_IF
		IF  ARiStnManualUSSideBsv[iStnFL] > 100 THEN ARiStnManualUSSideBsv[iStnFL] := 100; ELSIF ARiStnManualUSSideBsv[iStnFL] < 10 THEN ARiStnManualUSSideBsv[iStnFL] := 10; END_IF
		IF  ARiStnManualUSSideCsv[iStnFL] > 100 THEN ARiStnManualUSSideCsv[iStnFL] := 100; ELSIF ARiStnManualUSSideCsv[iStnFL] < 10 THEN ARiStnManualUSSideCsv[iStnFL] := 10; END_IF
		IF  ARiStnManualUSSideDsv[iStnFL] > 100 THEN ARiStnManualUSSideDsv[iStnFL] := 100; ELSIF ARiStnManualUSSideDsv[iStnFL] < 10 THEN ARiStnManualUSSideDsv[iStnFL] := 10; END_IF

	END_IF
END_FOR

(*Blower Inverter Manual Hz Setting Control*) (*For Fix Frequency*)
(*=========================================================*)
iStnFL := 1;
FOR iStnFL := 1 TO iStnQty DO
	IF iStnFL >= 1 AND iStnFL <= iStnQty THEN

		IF  ARiStnManualBlowerInvPercentSV[iStnFL] > 100 THEN ARiStnManualBlowerInvPercentSV[iStnFL] := 100; ELSIF ARiStnManualBlowerInvPercentSV[iStnFL] < 40 THEN ARiStnManualBlowerInvPercentSV[iStnFL] := 40; END_IF

	END_IF
END_FOR


(*Station Dripping, StnArmDetectZoneRange, StnTolerance, Stn Water TopUp Ctrl*)
(*=========================================================*)
iStnFL := 1;
FOR iStnFL := 1 TO iStnQty DO
	IF iStnFL >= 1 AND iStnFL <= iStnQty THEN

